KUKA KRL program: MyProgram_027().src

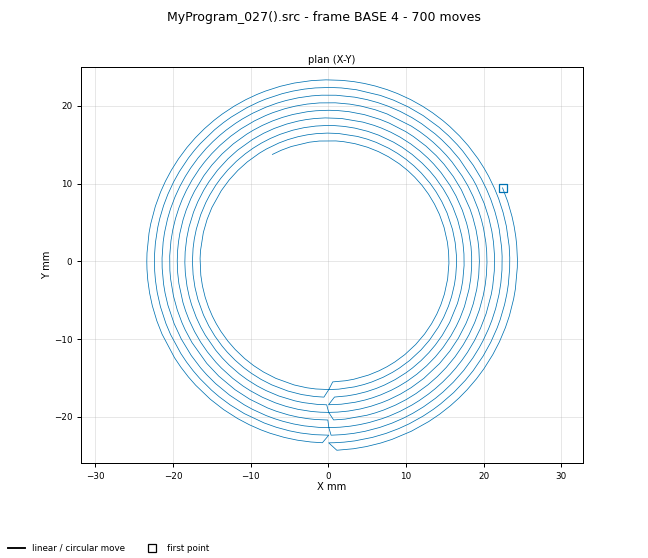
[picture p0: tool path of MyProgram_027().src in frame BASE 4, 700 of 700 moves have a stored position in this frame; points joined in program order, loops and branches not executed]
&ACCESS RVP
&REL 1
&PARAM TEMPLATE = C:\KRC\Roboter\Template\vorgabe
&PARAM EDITMASK = *
DEF MyProgram_027()
; ---- Setting reference (Base) ----
$BASE = BASE_DATA[4]

; --------------------------
; ---- Setting tool (TCP) ----
$TOOL = TOOL_DATA[3]
; --------------------------

$VEL.CP = VEL_APROX_PRINT
Startdeposition()
$VEL.CP = VEL_PRINT
LIN {X 22.4287,Y 9.4564,Z 58,A 14.1912,B 24.8124,C -3.1589,E1 25.1485,E2 -651.5768} C_DIS
LIN {X 23.1014,Y 7.6686,Z 58,A 9.7649,B 24.8138,C -3.1468,E1 25.1526,E2 -647.1466} C_DIS
LIN {X 23.6458,Y 5.7738,Z 58,A 5.5518,B 24.8149,C -3.1377,E1 25.1557,E2 -642.9363} C_DIS
LIN {X 23.9173,Y 4.5201,Z 58,A 2.5126,B 24.816,C -3.1284,E1 25.1574,E2 -639.8928} C_DIS
LIN {X 24.1337,Y 3.1677,Z 58,A -0.5395,B 24.8169,C -3.1205,E1 25.1586,E2 -636.8398} C_DIS
LIN {X 24.2489,Y 2.1152,Z 58,A -3.4554,B 24.8184,C -3.1081,E1 25.1594,E2 -633.9119} C_DIS
LIN {X 24.3395,Y 0.2898,Z 58,A -7.2887,B 24.8193,C -3.0999,E1 25.1598,E2 -630.082} C_DIS
LIN {X 24.3283,Y -0.7779,Z 58,A -10.7104,B 24.8214,C -3.082,E1 25.1595,E2 -626.6383} C_DIS
LIN {X 24.0781,Y -3.5664,Z 58,A -15.9759,B 24.8221,C -3.0762,E1 25.158,E2 -621.39} C_DIS
LIN {X 23.8573,Y -4.8272,Z 58,A -20.0449,B 24.8245,C -3.0551,E1 25.1558,E2 -617.295} C_DIS
LIN {X 23.313,Y -6.9977,Z 58,A -24.788,B 24.8257,C -3.0447,E1 25.1524,E2 -612.5545} C_DIS
LIN {X 22.7904,Y -8.5482,Z 58,A -28.7704,B 24.8272,C -3.0317,E1 25.1486,E2 -608.5636} C_DIS
LIN {X 22.0222,Y -10.3681,Z 58,A -33.8022,B 24.8293,C -3.0139,E1 25.1429,E2 -603.517} C_DIS
LIN {X 21.1792,Y -11.9952,Z 58,A -37.9863,B 24.8305,C -3.003,E1 25.1373,E2 -599.3291} C_DIS
LIN {X 20.022,Y -13.8417,Z 58,A -42.6404,B 24.8315,C -2.9941,E1 25.1302,E2 -594.677} C_DIS
LIN {X 19.0636,Y -15.1342,Z 58,A -46.5415,B 24.8328,C -2.983,E1 25.1235,E2 -590.7681} C_DIS
LIN {X 17.8586,Y -16.5394,Z 58,A -50.7568,B 24.8338,C -2.9737,E1 25.1157,E2 -586.5496} C_DIS
LIN {X 16.8309,Y -17.584,Z 58,A -54.1448,B 24.8346,C -2.9662,E1 25.109,E2 -583.1581} C_DIS
LIN {X 15.7146,Y -18.588,Z 58,A -57.8818,B 24.8358,C -2.9563,E1 25.1011,E2 -579.4124} C_DIS
LIN {X 14.3281,Y -19.6766,Z 58,A -61.9971,B 24.8367,C -2.9481,E1 25.0919,E2 -575.2925} C_DIS
LIN {X 12.9267,Y -20.6245,Z 58,A -66.2083,B 24.8377,C -2.9384,E1 25.082,E2 -571.072} C_DIS
LIN {X 10.6726,Y -21.8765,Z 58,A -72.7265,B 24.8393,C -2.9241,E1 25.0658,E2 -564.5382} C_DIS
LIN {X 8.2202,Y -22.9104,Z 58,A -78.0666,B 24.8393,C -2.9242,E1 25.052,E2 -559.2102} C_DIS
LIN {X 6.7478,Y -23.3869,Z 58,A -81.784,B 24.8398,C -2.9194,E1 25.0421,E2 -555.488} C_DIS
LIN {X 4.9064,Y -23.841,Z 58,A -86.3778,B 24.8404,C -2.9142,E1 25.0295,E2 -550.888} C_DIS
LIN {X 3.2399,Y -24.124,Z 58,A -90.0318,B 24.8404,C -2.9142,E1 25.0195,E2 -547.2376} C_DIS
LIN {X 1.0965,Y -24.316,Z 58,A -95.7147,B 24.8412,C -2.9068,E1 25.0036,E2 -541.5396} C_DIS
LIN {X 1.0965,Y -24.316,Z 58,A -95.7147,B 24.8412,C -2.9068,E1 25.0036,E2 -541.5396} C_DIS
Enddeposition()
LIN {X 0.0491,Y -23.3612,Z 58,A -97.7933,B 24.839,C -2.9266,E1 24.9979,E2 -539.5083} C_DIS
Startdeposition()
$VEL.CP = VEL_PRINT
LIN {X 0.753,Y -23.3494,Z 58,A -94.2208,B 24.8374,C -2.9419,E1 25.008,E2 -543.1168} C_DIS
LIN {X 2.0258,Y -23.2738,Z 58,A -91.3521,B 24.8374,C -2.9412,E1 25.016,E2 -545.9823} C_DIS
LIN {X 3.4162,Y -23.1102,Z 58,A -87.1337,B 24.8364,C -2.9501,E1 25.0277,E2 -550.2184} C_DIS
LIN {X 5.6877,Y -22.6583,Z 58,A -81.8177,B 24.8362,C -2.952,E1 25.0422,E2 -555.5318} C_DIS
LIN {X 7.425,Y -22.15,Z 58,A -77.4169,B 24.8357,C -2.9568,E1 25.0539,E2 -559.9358} C_DIS
LIN {X 9.059,Y -21.533,Z 58,A -73.7377,B 24.8357,C -2.957,E1 25.0634,E2 -563.6074} C_DIS
LIN {X 10.4154,Y -20.9112,Z 58,A -69.2878,B 24.8342,C -2.9701,E1 25.0747,E2 -568.0768} C_DIS
LIN {X 12.2027,Y -19.9213,Z 58,A -64.5258,B 24.8335,C -2.9765,E1 25.0862,E2 -572.8396} C_DIS
LIN {X 13.4975,Y -19.0679,Z 58,A -60.5918,B 24.8325,C -2.9852,E1 25.0953,E2 -576.7809} C_DIS
LIN {X 14.4357,Y -18.3677,Z 58,A -57.4005,B 24.8315,C -2.9945,E1 25.1023,E2 -579.9824} C_DIS
LIN {X 16.1336,Y -16.8961,Z 58,A -52.2089,B 24.8304,C -3.0037,E1 25.113,E2 -585.1748} C_DIS
LIN {X 17.6418,Y -15.3144,Z 58,A -47.4897,B 24.8297,C -3.0102,E1 25.1219,E2 -589.8886} C_DIS
LIN {X 18.6459,Y -14.0745,Z 58,A -42.8116,B 24.8276,C -3.0283,E1 25.13,E2 -594.5878} C_DIS
LIN {X 19.9336,Y -12.1826,Z 58,A -37.1639,B 24.8258,C -3.0441,E1 25.1386,E2 -600.2444} C_DIS
LIN {X 20.9152,Y -10.4066,Z 58,A -32.457,B 24.8245,C -3.0554,E1 25.1446,E2 -604.9534} C_DIS
LIN {X 21.729,Y -8.5794,Z 58,A -28.1395,B 24.8236,C -3.0635,E1 25.1494,E2 -609.2665} C_DIS
LIN {X 22.1157,Y -7.5274,Z 58,A -25.0112,B 24.8221,C -3.076,E1 25.1522,E2 -612.4065} C_DIS
LIN {X 22.6865,Y -5.5752,Z 58,A -20.1081,B 24.8205,C -3.0903,E1 25.1558,E2 -617.3155} C_DIS
LIN {X 22.9834,Y -4.1863,Z 58,A -16.5509,B 24.8191,C -3.1019,E1 25.1577,E2 -620.8794} C_DIS
LIN {X 23.1698,Y -2.9863,Z 58,A -13.4153,B 24.8178,C -3.1129,E1 25.1589,E2 -624.0226} C_DIS
LIN {X 23.3426,Y -0.9395,Z 58,A -8.919,B 24.8167,C -3.1227,E1 25.1597,E2 -628.5154} C_DIS
LIN {X 23.3568,Y 0.4688,Z 58,A -5.3427,B 24.8152,C -3.1348,E1 25.1597,E2 -632.0991} C_DIS
LIN {X 23.2798,Y 1.9538,Z 58,A -1.238,B 24.8133,C -3.1511,E1 25.1588,E2 -636.218} C_DIS
LIN {X 22.9166,Y 4.5391,Z 58,A 4.2783,B 24.8121,C -3.1609,E1 25.1564,E2 -641.7252} C_DIS
LIN {X 22.4933,Y 6.31,Z 58,A 9.6251,B 24.8094,C -3.1837,E1 25.1527,E2 -647.0951} C_DIS
LIN {X 21.9201,Y 8.0793,Z 58,A 13.523,B 24.8087,C -3.1897,E1 25.1491,E2 -650.9852} C_DIS
LIN {X 21.3892,Y 9.3949,Z 58,A 17.0683,B 24.8074,C -3.2001,E1 25.1452,E2 -654.5357} C_DIS
LIN {X 20.6396,Y 10.9433,Z 58,A 21.0402,B 24.8064,C -3.2088,E1 25.1403,E2 -658.5072} C_DIS
LIN {X 20.0488,Y 11.992,Z 58,A 24.1699,B 24.8052,C -3.2183,E1 25.1359,E2 -661.6433} C_DIS
LIN {X 19.2723,Y 13.2041,Z 58,A 28.0452,B 24.8037,C -3.2306,E1 25.1298,E2 -665.5285} C_DIS
LIN {X 18.0172,Y 14.871,Z 58,A 32.6958,B 24.8028,C -3.2378,E1 25.1218,E2 -670.1742} C_DIS
LIN {X 16.8934,Y 16.1364,Z 58,A 37.2521,B 24.8012,C -3.2508,E1 25.1132,E2 -674.7413} C_DIS
LIN {X 15.6106,Y 17.3802,Z 58,A 41.0651,B 24.8008,C -3.2539,E1 25.1054,E2 -678.5461} C_DIS
LIN {X 14.7291,Y 18.1332,Z 58,A 44.1503,B 24.7999,C -3.2614,E1 25.0988,E2 -681.6374} C_DIS
LIN {X 13.4156,Y 19.1256,Z 58,A 48.0828,B 24.7992,C -3.2672,E1 25.0899,E2 -685.5697} C_DIS
LIN {X 12.1321,Y 19.9642,Z 58,A 51.8621,B 24.7985,C -3.273,E1 25.081,E2 -689.3507} C_DIS
LIN {X 10.5843,Y 20.8263,Z 58,A 56.5365,B 24.7974,C -3.2816,E1 25.0694,E2 -694.0322} C_DIS
LIN {X 8.9243,Y 21.5896,Z 58,A 60.8731,B 24.797,C -3.2851,E1 25.0583,E2 -698.3666} C_DIS
LIN {X 7.5693,Y 22.1011,Z 58,A 64.2683,B 24.7968,C -3.2868,E1 25.0494,E2 -701.7589} C_DIS
LIN {X 6.0229,Y 22.5716,Z 58,A 68.0624,B 24.7966,C -3.288,E1 25.0393,E2 -705.5495} C_DIS
LIN {X 4.6413,Y 22.8959,Z 58,A 71.552,B 24.7964,C -3.2897,E1 25.0297,E2 -709.0387} C_DIS
LIN {X 3.3103,Y 23.1258,Z 58,A 74.9008,B 24.7963,C -3.291,E1 25.0205,E2 -712.3873} C_DIS
LIN {X 1.8029,Y 23.2918,Z 58,A 79.0541,B 24.7958,C -3.2947,E1 25.0089,E2 -716.5471} C_DIS
LIN {X -0.2978,Y 23.3597,Z 58,A 84.0444,B 24.796,C -3.2926,E1 24.995,E2 -721.5319} C_DIS
LIN {X -2.16,Y 23.2614,Z 58,A 88.9205,B 24.796,C -3.2929,E1 24.9814,E2 -726.4107} C_DIS
LIN {X -4.3701,Y 22.9492,Z 58,A 94.1198,B 24.7967,C -3.2872,E1 24.9671,E2 -731.601} C_DIS
LIN {X -6.1836,Y 22.5282,Z 58,A 98.7838,B 24.7972,C -3.2835,E1 24.9545,E2 -736.263} C_DIS
LIN {X -8.1141,Y 21.9067,Z 58,A 103.4711,B 24.7982,C -3.2757,E1 24.9422,E2 -740.9406} C_DIS
LIN {X -9.2066,Y 21.4713,Z 58,A 106.4345,B 24.7986,C -3.2722,E1 24.9345,E2 -743.9025} C_DIS
LIN {X -10.609,Y 20.8137,Z 58,A 110.0922,B 24.7994,C -3.2655,E1 24.9254,E2 -747.5537} C_DIS
LIN {X -12.0964,Y 19.9859,Z 58,A 114.7123,B 24.8,C -3.2609,E1 24.9142,E2 -752.1767} C_DIS
LIN {X -13.6533,Y 18.9565,Z 58,A 118.5178,B 24.8016,C -3.2477,E1 24.9055,E2 -755.9633} C_DIS
LIN {X -14.6701,Y 18.1811,Z 58,A 122.2839,B 24.802,C -3.2447,E1 24.8972,E2 -759.7362} C_DIS
LIN {X -15.9382,Y 17.0802,Z 58,A 126.4482,B 24.8031,C -3.2358,E1 24.8886,E2 -763.8958} C_DIS
LIN {X -17.1134,Y 15.9031,Z 58,A 130.3724,B 24.8044,C -3.2253,E1 24.881,E2 -767.8117} C_DIS
LIN {X -18.1978,Y 14.649,Z 58,A 134.5254,B 24.8055,C -3.2155,E1 24.8736,E2 -771.9605} C_DIS
LIN {X -19.2941,Y 13.1713,Z 58,A 139.5365,B 24.8067,C -3.2061,E1 24.8655,E2 -776.9735} C_DIS
LIN {X -20.1991,Y 11.7375,Z 58,A 143.4691,B 24.8082,C -3.1934,E1 24.8599,E2 -780.8961} C_DIS
LIN {X -20.9677,Y 10.3014,Z 58,A 147.0142,B 24.8099,C -3.1798,E1 24.8554,E2 -784.4276} C_DIS
LIN {X -21.5908,Y 8.9216,Z 58,A 151.509,B 24.8107,C -3.1727,E1 24.8504,E2 -788.9301} C_DIS
LIN {X -22.265,Y 7.0731,Z 58,A 156.3218,B 24.8125,C -3.1581,E1 24.8461,E2 -793.7354} C_DIS
LIN {X -22.8563,Y 4.8334,Z 58,A 161.8894,B 24.8146,C -3.1401,E1 24.8425,E2 -799.2925} C_DIS
LIN {X -23.0779,Y 3.6294,Z 58,A 165.278,B 24.8155,C -3.1326,E1 24.8411,E2 -802.6833} C_DIS
LIN {X -23.337,Y 1.0643,Z 58,A 170.5929,B 24.8184,C -3.1082,E1 24.8399,E2 -807.9716} C_DIS
LIN {X -23.3617,Y -0.0144,Z 58,A 173.2645,B 24.8193,C -3.1,E1 24.8398,E2 -810.6398} C_DIS
LIN {X -23.3392,Y -1.02,Z 58,A 175.8052,B 24.8202,C -3.0927,E1 24.84,E2 -813.1783} C_DIS
LIN {X -23.2364,Y -2.414,Z 58,A 179.6817,B 24.8212,C -3.0843,E1 24.841,E2 -817.0578} C_DIS
LIN {X -23.0029,Y -4.0772,Z 58,A -176.121,B 24.8226,C -3.0721,E1 24.8428,E2 -821.251} C_DIS
LIN {X -22.6514,Y -5.7166,Z 58,A -171.9113,B 24.8239,C -3.0603,E1 24.8455,E2 -825.4571} C_DIS
LIN {X -22.0687,Y -7.664,Z 58,A -166.7853,B 24.8255,C -3.0466,E1 24.8499,E2 -830.5795} C_DIS
LIN {X -21.4015,Y -9.3668,Z 58,A -161.5782,B 24.8265,C -3.0378,E1 24.8556,E2 -835.7944} C_DIS
LIN {X -19.7861,Y -12.4207,Z 58,A -154.6271,B 24.83,C -3.0077,E1 24.865,E2 -842.7098} C_DIS
LIN {X -18.9703,Y -13.6339,Z 58,A -150.229,B 24.8305,C -3.0033,E1 24.872,E2 -847.1192} C_DIS
LIN {X -18.0166,Y -14.8715,Z 58,A -146.7524,B 24.8317,C -2.9925,E1 24.8781,E2 -850.5863} C_DIS
LIN {X -17.0625,Y -15.9571,Z 58,A -142.5184,B 24.8321,C -2.9888,E1 24.8861,E2 -854.8302} C_DIS
LIN {X -15.1815,Y -17.7562,Z 58,A -136.8493,B 24.834,C -2.9722,E1 24.8977,E2 -860.4824} C_DIS
LIN {X -13.4696,Y -19.0872,Z 58,A -130.4927,B 24.8343,C -2.9697,E1 24.912,E2 -866.8557} C_DIS
LIN {X -11.6792,Y -20.2323,Z 58,A -126.0931,B 24.8357,C -2.957,E1 24.9224,E2 -871.2386} C_DIS
LIN {X -10.1604,Y -21.0363,Z 58,A -122.0125,B 24.8363,C -2.951,E1 24.9326,E2 -875.3159} C_DIS
LIN {X -8.6852,Y -21.6874,Z 58,A -118.3884,B 24.837,C -2.9447,E1 24.9418,E2 -878.9333} C_DIS
LIN {X -7.4925,Y -22.1274,Z 58,A -114.5721,B 24.8368,C -2.947,E1 24.9519,E2 -882.7627} C_DIS
LIN {X -5.6895,Y -22.6585,Z 58,A -110.4971,B 24.8375,C -2.9403,E1 24.9629,E2 -886.8281} C_DIS
LIN {X -4.0034,Y -23.0159,Z 58,A -105.4321,B 24.837,C -2.945,E1 24.9768,E2 -891.9099} C_DIS
LIN {X -2.2388,Y -23.2541,Z 58,A -101.6737,B 24.8376,C -2.9397,E1 24.9872,E2 -895.6581} C_DIS
LIN {X -0.7601,Y -23.3492,Z 58,A -97.8291,B 24.8374,C -2.9417,E1 24.9979,E2 -899.5083} C_DIS
LIN {X -0.7601,Y -23.3492,Z 58,A -97.8291,B 24.8374,C -2.9417,E1 24.9979,E2 -899.5083} C_DIS
Enddeposition()
LIN {X 0.0594,Y -22.3764,Z 58,A -97.5822,B 24.837,C -2.9453,E1 24.9986,E2 -899.7639} C_DIS
Startdeposition()
$VEL.CP = VEL_PRINT
LIN {X -1.7887,Y -22.3107,Z 58,A -102.6934,B 24.8373,C -2.9422,E1 24.9844,E2 -894.6438} C_DIS
LIN {X -3.5725,Y -22.0957,Z 58,A -107.3153,B 24.8373,C -2.943,E1 24.9716,E2 -890.0201} C_DIS
LIN {X -4.9833,Y -21.8206,Z 58,A -110.5248,B 24.8367,C -2.9478,E1 24.9628,E2 -886.8182} C_DIS
LIN {X -6.6868,Y -21.3602,Z 58,A -116.1215,B 24.8372,C -2.9436,E1 24.9478,E2 -881.2024} C_DIS
LIN {X -8.2481,Y -20.8072,Z 58,A -120.6031,B 24.8369,C -2.946,E1 24.9361,E2 -876.7169} C_DIS
LIN {X -10.8134,Y -19.5971,Z 58,A -126.9982,B 24.8353,C -2.96,E1 24.9202,E2 -870.3379} C_DIS
LIN {X -12.6262,Y -18.4813,Z 58,A -133.0282,B 24.8348,C -2.9649,E1 24.9061,E2 -864.3002} C_DIS
LIN {X -14.016,Y -17.4505,Z 58,A -136.4557,B 24.8333,C -2.9781,E1 24.8986,E2 -860.8916} C_DIS
LIN {X -15.0383,Y -16.5769,Z 58,A -140.5893,B 24.833,C -2.9809,E1 24.8899,E2 -856.7484} C_DIS
LIN {X -16.5556,Y -15.0627,Z 58,A -145.4598,B 24.8314,C -2.9955,E1 24.8805,E2 -851.8918} C_DIS
LIN {X -17.4052,Y -14.0722,Z 58,A -149.0695,B 24.8307,C -3.0017,E1 24.874,E2 -848.2803} C_DIS
LIN {X -18.2465,Y -12.9621,Z 58,A -152.5872,B 24.8297,C -3.0104,E1 24.8682,E2 -844.7665} C_DIS
LIN {X -18.9806,Y -11.8619,Z 58,A -156.8774,B 24.8292,C -3.0146,E1 24.8617,E2 -840.4647} C_DIS
LIN {X -20.3019,Y -9.4219,Z 58,A -163.3655,B 24.8267,C -3.0364,E1 24.8535,E2 -833.994} C_DIS
LIN {X -20.8927,Y -8.0277,Z 58,A -167.7212,B 24.8257,C -3.0452,E1 24.849,E2 -829.6351} C_DIS
LIN {X -21.613,Y -5.8178,Z 58,A -172.7995,B 24.8232,C -3.0663,E1 24.8449,E2 -824.5779} C_DIS
LIN {X -22.0246,Y -3.9859,Z 58,A -178.1948,B 24.8219,C -3.0782,E1 24.8418,E2 -819.1796} C_DIS
LIN {X -22.2472,Y -2.4581,Z 58,A 178.0676,B 24.8204,C -3.0912,E1 24.8405,E2 -815.4506} C_DIS
LIN {X -22.3486,Y -1.2274,Z 58,A 174.5283,B 24.8194,C -3.0994,E1 24.8399,E2 -811.9098} C_DIS
LIN {X -22.3659,Y 0.8536,Z 58,A 169.598,B 24.8173,C -3.1176,E1 24.8399,E2 -806.9933} C_DIS
LIN {X -22.2556,Y 2.3786,Z 58,A 165.1888,B 24.8161,C -3.1278,E1 24.8411,E2 -802.5821} C_DIS
LIN {X -21.9494,Y 4.382,Z 58,A 160.6412,B 24.8138,C -3.1465,E1 24.8432,E2 -798.0523} C_DIS
LIN {X -21.681,Y 5.5591,Z 58,A 157.1953,B 24.8129,C -3.1545,E1 24.8455,E2 -794.6055} C_DIS
LIN {X -21.2056,Y 7.1618,Z 58,A 152.9812,B 24.8113,C -3.1678,E1 24.849,E2 -790.3989} C_DIS
LIN {X -20.6553,Y 8.6217,Z 58,A 148.825,B 24.81,C -3.1789,E1 24.8533,E2 -786.2461} C_DIS
LIN {X -19.9176,Y 10.2106,Z 58,A 143.8606,B 24.8087,C -3.1898,E1 24.8593,E2 -781.281} C_DIS
LIN {X -19.1663,Y 11.5597,Z 58,A 139.9008,B 24.8073,C -3.2008,E1 24.865,E2 -777.3269} C_DIS
LIN {X -17.9987,Y 13.3051,Z 58,A 135.1411,B 24.8053,C -3.2178,E1 24.8725,E2 -772.5847} C_DIS
LIN {X -17.2488,Y 14.2633,Z 58,A 132.085,B 24.8043,C -3.2261,E1 24.8778,E2 -769.534} C_DIS
LIN {X -16.4585,Y 15.1687,Z 58,A 127.8731,B 24.804,C -3.2282,E1 24.8858,E2 -765.3085} C_DIS
LIN {X -14.6393,Y 16.9314,Z 58,A 122.0959,B 24.8018,C -3.2462,E1 24.8976,E2 -759.5511} C_DIS
LIN {X -13.4935,Y 17.8577,Z 58,A 118.4161,B 24.8008,C -3.2545,E1 24.9057,E2 -755.8775} C_DIS
LIN {X -12.501,Y 18.566,Z 58,A 114.5849,B 24.8005,C -3.2568,E1 24.9146,E2 -752.0389} C_DIS
LIN {X -10.4803,Y 19.7772,Z 58,A 109.1764,B 24.7988,C -3.2704,E1 24.9276,E2 -746.6472} C_DIS
LIN {X -9.0313,Y 20.4796,Z 58,A 105.3376,B 24.7978,C -3.2782,E1 24.9373,E2 -742.8173} C_DIS
LIN {X -8.0558,Y 20.8828,Z 58,A 101.9318,B 24.7979,C -3.2776,E1 24.9462,E2 -739.4028} C_DIS
LIN {X -5.9481,Y 21.5771,Z 58,A 96.8474,B 24.7967,C -3.2875,E1 24.9597,E2 -734.3332} C_DIS
LIN {X -4.5409,Y 21.9167,Z 58,A 92.9641,B 24.7964,C -3.2896,E1 24.9703,E2 -730.4499} C_DIS
LIN {X -3.0809,Y 22.1694,Z 58,A 89.0937,B 24.7962,C -3.2916,E1 24.981,E2 -726.5809} C_DIS
LIN {X -1.6805,Y 22.3194,Z 58,A 85.2928,B 24.7962,C -3.292,E1 24.9915,E2 -722.779} C_DIS
LIN {X 0.2375,Y 22.3811,Z 58,A 80.7154,B 24.7957,C -3.2955,E1 25.0043,E2 -718.2098} C_DIS
LIN {X 1.6744,Y 22.3198,Z 58,A 76.9456,B 24.7957,C -3.2949,E1 25.0148,E2 -714.44} C_DIS
LIN {X 3.6228,Y 22.0866,Z 58,A 70.9029,B 24.7969,C -3.2861,E1 25.0315,E2 -708.3818} C_DIS
LIN {X 6.6984,Y 21.3562,Z 58,A 63.2106,B 24.7971,C -3.2842,E1 25.0522,E2 -700.6972} C_DIS
LIN {X 8.4,Y 20.7463,Z 58,A 59.4451,B 24.7968,C -3.2869,E1 25.062,E2 -696.9462} C_DIS
LIN {X 10.3058,Y 19.8686,Z 58,A 52.692,B 24.799,C -3.2689,E1 25.079,E2 -690.1685} C_DIS
LIN {X 12.2114,Y 18.758,Z 58,A 47.4398,B 24.7996,C -3.2639,E1 25.0914,E2 -684.9211} C_DIS
LIN {X 14.2392,Y 17.269,Z 58,A 41.6217,B 24.8003,C -3.2582,E1 25.1042,E2 -679.1109} C_DIS
LIN {X 15.472,Y 16.1738,Z 58,A 37.5824,B 24.8011,C -3.2516,E1 25.1125,E2 -675.0722} C_DIS
LIN {X 16.6049,Y 15.0081,Z 58,A 33.7383,B 24.8019,C -3.2457,E1 25.1199,E2 -671.2309} C_DIS
LIN {X 17.3174,Y 14.1806,Z 58,A 30.4374,B 24.8032,C -3.2346,E1 25.1258,E2 -667.9188} C_DIS
LIN {X 18.6592,Y 12.3614,Z 58,A 24.2702,B 24.8054,C -3.2169,E1 25.1357,E2 -661.7396} C_DIS
LIN {X 19.684,Y 10.6539,Z 58,A 19.7371,B 24.8063,C -3.2091,E1 25.142,E2 -657.2117} C_DIS
LIN {X 20.3685,Y 9.2781,Z 58,A 16.0112,B 24.8074,C -3.2005,E1 25.1464,E2 -653.4853} C_DIS
LIN {X 20.9171,Y 7.9652,Z 58,A 12.3886,B 24.8086,C -3.1904,E1 25.1502,E2 -649.859} C_DIS
LIN {X 21.4372,Y 6.436,Z 58,A 8.0462,B 24.8103,C -3.1763,E1 25.1539,E2 -645.5077} C_DIS
LIN {X 21.7836,Y 5.1424,Z 58,A 5.1065,B 24.8109,C -3.1711,E1 25.1559,E2 -642.5728} C_DIS
LIN {X 21.9951,Y 4.1454,Z 58,A 1.6107,B 24.8129,C -3.1541,E1 25.1578,E2 -639.0571} C_DIS
LIN {X 22.3104,Y 1.7924,Z 58,A -3.5855,B 24.8141,C -3.1446,E1 25.1594,E2 -633.869} C_DIS
LIN {X 22.373,Y 0.6481,Z 58,A -6.8291,B 24.8155,C -3.1323,E1 25.1598,E2 -630.6154} C_DIS
LIN {X 22.3556,Y -1.1014,Z 58,A -10.8962,B 24.8167,C -3.1226,E1 25.1595,E2 -626.5495} C_DIS
LIN {X 22.2102,Y -2.7725,Z 58,A -15.339,B 24.8184,C -3.1076,E1 25.1582,E2 -622.0977} C_DIS
LIN {X 21.9749,Y -4.251,Z 58,A -19.4147,B 24.8201,C -3.0932,E1 25.1563,E2 -618.0116} C_DIS
LIN {X 21.5448,Y -6.0656,Z 58,A -23.856,B 24.8214,C -3.082,E1 25.1532,E2 -613.5693} C_DIS
LIN {X 21.0614,Y -7.5761,Z 58,A -28.0424,B 24.823,C -3.0684,E1 25.1495,E2 -609.3744} C_DIS
LIN {X 20.6289,Y -8.683,Z 58,A -31.1464,B 24.8241,C -3.0587,E1 25.1462,E2 -606.2646} C_DIS
LIN {X 19.9077,Y -10.2301,Z 58,A -35.0818,B 24.8251,C -3.0505,E1 25.1414,E2 -602.3309} C_DIS
LIN {X 19.4242,Y -11.1207,Z 58,A -38.0233,B 24.8263,C -3.0396,E1 25.1373,E2 -599.3789} C_DIS
LIN {X 18.6136,Y -12.4304,Z 58,A -42.1385,B 24.8278,C -3.0271,E1 25.1311,E2 -595.2547} C_DIS
LIN {X 17.4263,Y -14.0461,Z 58,A -46.9358,B 24.8289,C -3.017,E1 25.123,E2 -590.4562} C_DIS
LIN {X 16.0944,Y -15.554,Z 58,A -52.29,B 24.8306,C -3.0024,E1 25.1129,E2 -585.0911} C_DIS
LIN {X 14.7617,Y -16.824,Z 58,A -57.1683,B 24.832,C -2.9902,E1 25.1028,E2 -580.2034} C_DIS
LIN {X 13.7674,Y -17.6476,Z 58,A -60.2302,B 24.8325,C -2.9854,E1 25.0961,E2 -577.1417} C_DIS
LIN {X 12.2563,Y -18.7283,Z 58,A -65.0156,B 24.8336,C -2.9759,E1 25.085,E2 -572.35} C_DIS
LIN {X 10.8816,Y -19.5592,Z 58,A -68.887,B 24.8341,C -2.9708,E1 25.0757,E2 -568.4783} C_DIS
LIN {X 9.6925,Y -20.1748,Z 58,A -72.1113,B 24.8345,C -2.9672,E1 25.0676,E2 -565.254} C_DIS
LIN {X 8.1975,Y -20.8271,Z 58,A -77.0054,B 24.8359,C -2.9551,E1 25.055,E2 -560.3425} C_DIS
LIN {X 6.6205,Y -21.3808,Z 58,A -80.9282,B 24.8361,C -2.953,E1 25.0446,E2 -556.4223} C_DIS
LIN {X 4.7408,Y -21.8745,Z 58,A -86.0433,B 24.8368,C -2.9472,E1 25.0307,E2 -551.3005} C_DIS
LIN {X 3.2782,Y -22.1409,Z 58,A -89.3041,B 24.8366,C -2.9488,E1 25.0217,E2 -548.0468} C_DIS
LIN {X 1.843,Y -22.3064,Z 58,A -92.8669,B 24.8367,C -2.9478,E1 25.0118,E2 -544.4841} C_DIS
LIN {X 0.3571,Y -22.3795,Z 58,A -97.5689,B 24.8376,C -2.9398,E1 24.9986,E2 -539.7639} C_DIS
LIN {X 0.3571,Y -22.3795,Z 58,A -97.5689,B 24.8376,C -2.9398,E1 24.9986,E2 -539.7639} C_DIS
Enddeposition()
LIN {X 0.0693,Y -21.4022,Z 58,A -96.3339,B 24.8341,C -2.9713,E1 25.0023,E2 -541.074} C_DIS
Startdeposition()
$VEL.CP = VEL_PRINT
LIN {X 1.5198,Y -21.3493,Z 58,A -91.7701,B 24.8333,C -2.9779,E1 25.0151,E2 -545.652} C_DIS
LIN {X 2.8494,Y -21.2129,Z 58,A -88.6846,B 24.8335,C -2.9762,E1 25.0236,E2 -548.7311} C_DIS
LIN {X 4.0899,Y -21.0073,Z 58,A -85.405,B 24.8333,C -2.9782,E1 25.0326,E2 -552.0118} C_DIS
LIN {X 5.2662,Y -20.7452,Z 58,A -81.7581,B 24.8326,C -2.9846,E1 25.0425,E2 -555.6688} C_DIS
LIN {X 6.9059,Y -20.2584,Z 58,A -77.6775,B 24.8325,C -2.9857,E1 25.0534,E2 -559.7446} C_DIS
LIN {X 7.8829,Y -19.8986,Z 58,A -74.7362,B 24.8319,C -2.9907,E1 25.0611,E2 -562.6914} C_DIS
LIN {X 9.2231,Y -19.314,Z 58,A -70.3467,B 24.8308,C -3.0007,E1 25.0723,E2 -567.0936} C_DIS
LIN {X 10.7484,Y -18.5088,Z 58,A -66.2126,B 24.8304,C -3.0043,E1 25.0824,E2 -571.2242} C_DIS
LIN {X 11.7,Y -17.9216,Z 58,A -63.1037,B 24.8296,C -3.0109,E1 25.0897,E2 -574.3388} C_DIS
LIN {X 12.8554,Y -17.1124,Z 58,A -59.4843,B 24.8289,C -3.0171,E1 25.0979,E2 -577.9599} C_DIS
LIN {X 13.7488,Y -16.403,Z 58,A -56.3175,B 24.828,C -3.0247,E1 25.1048,E2 -581.1328} C_DIS
LIN {X 14.7388,Y -15.5201,Z 58,A -52.7543,B 24.8271,C -3.0329,E1 25.1121,E2 -584.701} C_DIS
LIN {X 15.6931,Y -14.5536,Z 58,A -49.3674,B 24.8264,C -3.0392,E1 25.1186,E2 -588.0883} C_DIS
LIN {X 16.4198,Y -13.7291,Z 58,A -46.2674,B 24.8253,C -3.0482,E1 25.1243,E2 -591.1954} C_DIS
LIN {X 17.2074,Y -12.7282,Z 58,A -42.9241,B 24.8244,C -3.0564,E1 25.1299,E2 -594.5423} C_DIS
LIN {X 17.9074,Y -11.7228,Z 58,A -39.2492,B 24.8229,C -3.0692,E1 25.1357,E2 -598.2294} C_DIS
LIN {X 18.8206,Y -10.1922,Z 58,A -34.6991,B 24.8216,C -3.0805,E1 25.142,E2 -602.7826} C_DIS
LIN {X 19.5937,Y -8.6123,Z 58,A -29.3344,B 24.8192,C -3.1009,E1 25.1482,E2 -608.1666} C_DIS
LIN {X 20.3118,Y -6.7471,Z 58,A -23.9701,B 24.8173,C -3.1171,E1 25.1532,E2 -613.5393} C_DIS
LIN {X 20.9731,Y -4.2692,Z 58,A -18.2317,B 24.8162,C -3.1266,E1 25.157,E2 -619.267} C_DIS
LIN {X 21.1564,Y -3.2408,Z 58,A -14.9725,B 24.8146,C -3.1401,E1 25.1584,E2 -622.5389} C_DIS
LIN {X 21.3682,Y -1.2241,Z 58,A -9.2908,B 24.8123,C -3.1597,E1 25.1597,E2 -628.2333} C_DIS
LIN {X 21.3873,Y 0.8276,Z 58,A -4.2264,B 24.8108,C -3.1723,E1 25.1595,E2 -633.2975} C_DIS
LIN {X 21.2582,Y 2.4869,Z 58,A 0.2319,B 24.8091,C -3.1861,E1 25.1583,E2 -637.7621} C_DIS
LIN {X 21.0478,Y 3.8847,Z 58,A 3.6058,B 24.8082,C -3.1934,E1 25.1567,E2 -641.1334} C_DIS
LIN {X 20.665,Y 5.5726,Z 58,A 9.342,B 24.8052,C -3.2183,E1 25.1528,E2 -646.8957} C_DIS
LIN {X 20.069,Y 7.4386,Z 58,A 14.4314,B 24.8036,C -3.2318,E1 25.1481,E2 -651.9884} C_DIS
LIN {X 19.0671,Y 9.7232,Z 58,A 19.9812,B 24.8027,C -3.2389,E1 25.1416,E2 -657.525} C_DIS
LIN {X 18.6099,Y 10.5724,Z 58,A 23.8934,B 24.8003,C -3.2586,E1 25.1361,E2 -661.4638} C_DIS
LIN {X 16.8781,Y 13.1612,Z 58,A 31.1716,B 24.799,C -3.2686,E1 25.1244,E2 -668.7301} C_DIS
LIN {X 15.6725,Y 14.5761,Z 58,A 36.4374,B 24.7973,C -3.2822,E1 25.1146,E2 -674.0048} C_DIS
LIN {X 14.6343,Y 15.6184,Z 58,A 40.2325,B 24.7965,C -3.2888,E1 25.107,E2 -677.7997} C_DIS
LIN {X 13.7487,Y 16.4035,Z 58,A 43.6494,B 24.7955,C -3.2969,E1 25.0997,E2 -681.2228} C_DIS
LIN {X 12.0117,Y 17.7147,Z 58,A 48.9825,B 24.7948,C -3.3023,E1 25.0876,E2 -686.5498} C_DIS
LIN {X 10.7598,Y 18.5017,Z 58,A 52.8179,B 24.7943,C -3.3069,E1 25.0785,E2 -690.3843} C_DIS
LIN {X 9.2573,Y 19.2976,Z 58,A 58.1125,B 24.7928,C -3.3187,E1 25.0652,E2 -695.6925} C_DIS
LIN {X 7.6976,Y 19.9713,Z 58,A 62.0521,B 24.7928,C -3.3182,E1 25.0551,E2 -699.6221} C_DIS
LIN {X 6.3869,Y 20.4277,Z 58,A 65.6538,B 24.7926,C -3.3203,E1 25.0455,E2 -703.2218} C_DIS
LIN {X 4.9912,Y 20.8132,Z 58,A 69.4819,B 24.7924,C -3.3222,E1 25.0352,E2 -707.0485} C_DIS
LIN {X 3.3995,Y 21.1316,Z 58,A 74.5674,B 24.7915,C -3.3293,E1 25.0212,E2 -712.1454} C_DIS
LIN {X 1.0071,Y 21.3796,Z 58,A 80.93,B 24.7915,C -3.329,E1 25.0035,E2 -718.5042} C_DIS
LIN {X -0.8511,Y 21.3863,Z 58,A 85.1036,B 24.7923,C -3.3223,E1 24.9919,E2 -722.662} C_DIS
LIN {X -2.12,Y 21.2982,Z 58,A 89.072,B 24.7921,C -3.3244,E1 24.9808,E2 -726.6375} C_DIS
LIN {X -3.8656,Y 21.0513,Z 58,A 93.663,B 24.7926,C -3.3204,E1 24.9682,E2 -731.2229} C_DIS
LIN {X -5.4449,Y 20.6991,Z 58,A 97.5083,B 24.7935,C -3.3134,E1 24.9578,E2 -735.057} C_DIS
LIN {X -6.6125,Y 20.3561,Z 58,A 101.0629,B 24.7937,C -3.3116,E1 24.9483,E2 -738.6134} C_DIS
LIN {X -8.0513,Y 19.8311,Z 58,A 105.4185,B 24.7942,C -3.3078,E1 24.9369,E2 -742.969} C_DIS
LIN {X -9.7406,Y 19.0582,Z 58,A 110.2465,B 24.7952,C -3.2994,E1 24.9248,E2 -747.7894} C_DIS
LIN {X -11.0483,Y 18.3307,Z 58,A 113.9019,B 24.7963,C -3.2906,E1 24.916,E2 -751.4348} C_DIS
LIN {X -11.947,Y 17.7586,Z 58,A 117.5019,B 24.7965,C -3.2892,E1 24.9076,E2 -755.0431} C_DIS
LIN {X -13.1313,Y 16.9018,Z 58,A 120.8139,B 24.7978,C -3.2782,E1 24.9002,E2 -758.3407} C_DIS
LIN {X -13.9343,Y 16.2461,Z 58,A 123.6422,B 24.7986,C -3.2725,E1 24.8942,E2 -761.1662} C_DIS
LIN {X -14.8529,Y 15.4106,Z 58,A 127.0044,B 24.7995,C -3.2652,E1 24.8873,E2 -764.5246} C_DIS
LIN {X -15.7184,Y 14.5269,Z 58,A 130.4415,B 24.8004,C -3.2578,E1 24.8807,E2 -767.9591} C_DIS
LIN {X -16.7726,Y 13.2957,Z 58,A 135.0521,B 24.8016,C -3.2481,E1 24.8725,E2 -772.5678} C_DIS
LIN {X -17.7086,Y 12.0208,Z 58,A 139.1812,B 24.803,C -3.2364,E1 24.8659,E2 -776.6891} C_DIS
LIN {X -18.4038,Y 10.927,Z 58,A 142.3461,B 24.8043,C -3.2256,E1 24.8613,E2 -779.8442} C_DIS
LIN {X -19.0851,Y 9.6879,Z 58,A 146.59,B 24.8054,C -3.2167,E1 24.8558,E2 -784.0896} C_DIS
LIN {X -19.7286,Y 8.2992,Z 58,A 150.5497,B 24.8069,C -3.2042,E1 24.8513,E2 -788.0409} C_DIS
LIN {X -20.3165,Y 6.7338,Z 58,A 154.7785,B 24.8087,C -3.1898,E1 24.8473,E2 -792.2592} C_DIS
LIN {X -20.6915,Y 5.474,Z 58,A 158.959,B 24.8096,C -3.1817,E1 24.8442,E2 -796.4446} C_DIS
LIN {X -21.0816,Y 3.6974,Z 58,A 163.3734,B 24.8116,C -3.1649,E1 24.8418,E2 -800.8446} C_DIS
LIN {X -21.2577,Y 2.4906,Z 58,A 167.1623,B 24.8126,C -3.1568,E1 24.8405,E2 -804.6369} C_DIS
LIN {X -21.3994,Y 0.402,Z 58,A 172.4761,B 24.8148,C -3.1382,E1 24.8398,E2 -809.938} C_DIS
LIN {X -21.3849,Y -0.8776,Z 58,A 176.3477,B 24.8159,C -3.1293,E1 24.8401,E2 -813.8118} C_DIS
LIN {X -21.2032,Y -2.9204,Z 58,A -178.7341,B 24.8181,C -3.1102,E1 24.8416,E2 -818.7135} C_DIS
LIN {X -21.0075,Y -4.0947,Z 58,A -175.2363,B 24.8191,C -3.1018,E1 24.8434,E2 -822.212} C_DIS
LIN {X -20.6458,Y -5.6437,Z 58,A -170.558,B 24.8204,C -3.091,E1 24.8466,E2 -826.8916} C_DIS
LIN {X -19.8389,Y -8.0321,Z 58,A -164.4138,B 24.8229,C -3.0691,E1 24.8524,E2 -833.0183} C_DIS
LIN {X -18.9192,Y -10.0068,Z 58,A -157.6316,B 24.8242,C -3.0576,E1 24.8608,E2 -839.8095} C_DIS
LIN {X -17.6345,Y -12.1284,Z 58,A -150.881,B 24.8261,C -3.0416,E1 24.8711,E2 -846.5558} C_DIS
LIN {X -16.4221,Y -13.7264,Z 58,A -146.525,B 24.8281,C -3.0243,E1 24.8786,E2 -850.8908} C_DIS
LIN {X -15.6668,Y -14.5823,Z 58,A -143.5566,B 24.8289,C -3.0173,E1 24.8842,E2 -853.8556} C_DIS
LIN {X -14.5057,Y -15.7379,Z 58,A -138.3999,B 24.8294,C -3.0125,E1 24.8946,E2 -859.0223} C_DIS
LIN {X -12.6922,Y -17.2334,Z 58,A -131.5397,B 24.8303,C -3.0047,E1 24.9097,E2 -865.8889} C_DIS
LIN {X -10.8237,Y -18.4648,Z 58,A -126.387,B 24.8318,C -2.9912,E1 24.9219,E2 -871.0254} C_DIS
LIN {X -9.7369,Y -19.0597,Z 58,A -122.9346,B 24.8322,C -2.9879,E1 24.9305,E2 -874.4794} C_DIS
LIN {X -7.9985,Y -19.8526,Z 58,A -118.2818,B 24.8331,C -2.9797,E1 24.9423,E2 -879.1238} C_DIS
LIN {X -6.9053,Y -20.2587,Z 58,A -115.1019,B 24.8334,C -2.9775,E1 24.9507,E2 -882.3047} C_DIS
LIN {X -5.8242,Y -20.5955,Z 58,A -112.1278,B 24.8337,C -2.9751,E1 24.9587,E2 -885.278} C_DIS
LIN {X -4.4547,Y -20.9347,Z 58,A -107.877,B 24.8335,C -2.9765,E1 24.9703,E2 -889.5376} C_DIS
LIN {X -3.0926,Y -21.1785,Z 58,A -104.2159,B 24.8336,C -2.9752,E1 24.9804,E2 -893.199} C_DIS
LIN {X -1.2575,Y -21.3663,Z 58,A -99.4586,B 24.8338,C -2.9737,E1 24.9936,E2 -897.955} C_DIS
LIN {X 0.0693,Y -21.4022,Z 58,A -97.6052,B 24.8351,C -2.962,E1 24.9987,E2 -899.7806} C_DIS
Enddeposition()
LIN {X 0.0693,Y -21.4022,Z 58,A -97.6052,B 24.8351,C -2.962,E1 24.9987,E2 -899.7806} C_DIS
Startdeposition()
$VEL.CP = VEL_PRINT
LIN {X -0.0586,Y -20.424,Z 58,A -98.287,B 24.8335,C -2.9769,E1 24.9969,E2 -899.1341} C_DIS
LIN {X -1.6552,Y -20.3567,Z 58,A -102.4124,B 24.8332,C -2.979,E1 24.9854,E2 -895.0127} C_DIS
LIN {X -2.7246,Y -20.2414,Z 58,A -105.6254,B 24.8333,C -2.9782,E1 24.9765,E2 -891.7956} C_DIS
LIN {X -3.9104,Y -20.0459,Z 58,A -108.963,B 24.8332,C -2.9795,E1 24.9673,E2 -888.4577} C_DIS
LIN {X -5.1213,Y -19.7715,Z 58,A -112.7276,B 24.8332,C -2.9796,E1 24.9571,E2 -884.6881} C_DIS
LIN {X -6.7102,Y -19.2901,Z 58,A -117.0919,B 24.8326,C -2.9848,E1 24.9455,E2 -880.3283} C_DIS
LIN {X -7.8166,Y -18.8693,Z 58,A -121.2762,B 24.8327,C -2.9831,E1 24.9346,E2 -876.1307} C_DIS
LIN {X -10.1008,Y -17.7516,Z 58,A -127.7286,B 24.8313,C -2.9956,E1 24.9187,E2 -869.6904} C_DIS
LIN {X -12.0003,Y -16.5256,Z 58,A -134.8567,B 24.8307,C -3.0016,E1 24.9022,E2 -862.5528} C_DIS
LIN {X -14.0953,Y -14.779,Z 58,A -143.2401,B 24.8294,C -3.0129,E1 24.8848,E2 -854.1631} C_DIS
LIN {X -15.6471,Y -13.1267,Z 58,A -149.7281,B 24.8278,C -3.0265,E1 24.873,E2 -847.678} C_DIS
LIN {X -17.5487,Y -10.4492,Z 58,A -157.6896,B 24.8246,C -3.0543,E1 24.8607,E2 -839.7431} C_DIS
LIN {X -18.4234,Y -8.8155,Z 58,A -162.3794,B 24.8228,C -3.0701,E1 24.8548,E2 -835.0663} C_DIS
LIN {X -18.8462,Y -7.8717,Z 58,A -165.7467,B 24.8221,C -3.0764,E1 24.851,E2 -831.6954} C_DIS
LIN {X -19.4425,Y -6.2548,Z 58,A -170.6189,B 24.8205,C -3.0901,E1 24.8466,E2 -826.8284} C_DIS
LIN {X -19.9345,Y -4.4434,Z 58,A -176.4767,B 24.8189,C -3.1037,E1 24.8427,E2 -820.9687} C_DIS
LIN {X -20.2972,Y -2.2732,Z 58,A 178.3183,B 24.8163,C -3.1258,E1 24.8406,E2 -815.7858} C_DIS
LIN {X -20.3898,Y -1.1818,Z 58,A 174.5621,B 24.8154,C -3.133,E1 24.8399,E2 -812.0242} C_DIS
LIN {X -20.412,Y 0.7019,Z 58,A 169.5522,B 24.8134,C -3.1504,E1 24.8399,E2 -807.0257} C_DIS
LIN {X -20.2541,Y 2.6291,Z 58,A 163.8252,B 24.8115,C -3.1662,E1 24.8416,E2 -801.3024} C_DIS
LIN {X -20.0148,Y 4.0678,Z 58,A 160.1309,B 24.8098,C -3.1802,E1 24.8435,E2 -797.6198} C_DIS
LIN {X -19.6661,Y 5.5125,Z 58,A 155.6043,B 24.8084,C -3.1917,E1 24.8466,E2 -793.0944} C_DIS
LIN {X -19.2249,Y 6.896,Z 58,A 151.7918,B 24.8068,C -3.2049,E1 24.8501,E2 -789.2918} C_DIS
LIN {X -18.7995,Y 7.9826,Z 58,A 148.612,B 24.8056,C -3.2149,E1 24.8534,E2 -786.1182} C_DIS
LIN {X -18.2634,Y 9.1429,Z 58,A 144.7735,B 24.8045,C -3.2244,E1 24.858,E2 -782.2815} C_DIS
LIN {X -17.5396,Y 10.4645,Z 58,A 140.2703,B 24.8031,C -3.2351,E1 24.8643,E2 -777.7806} C_DIS
LIN {X -16.5976,Y 11.9022,Z 58,A 135.8853,B 24.8014,C -3.2497,E1 24.8711,E2 -773.4089} C_DIS
LIN {X -15.9514,Y 12.7546,Z 58,A 132.6547,B 24.8005,C -3.2566,E1 24.8767,E2 -770.1793} C_DIS
LIN {X -15.0209,Y 13.8388,Z 58,A 128.7199,B 24.7993,C -3.2667,E1 24.884,E2 -766.2511} C_DIS
LIN {X -13.9341,Y 14.9327,Z 58,A 123.9175,B 24.7983,C -3.2746,E1 24.8936,E2 -761.4478} C_DIS
LIN {X -12.5691,Y 16.0986,Z 58,A 118.783,B 24.797,C -3.2849,E1 24.9047,E2 -756.3183} C_DIS
LIN {X -11.2286,Y 17.0604,Z 58,A 114.2023,B 24.7959,C -3.2939,E1 24.9152,E2 -751.744} C_DIS
LIN {X -9.4998,Y 18.0799,Z 58,A 108.6201,B 24.7947,C -3.3037,E1 24.9288,E2 -746.1689} C_DIS
LIN {X -8.069,Y 18.7626,Z 58,A 104.5369,B 24.7936,C -3.312,E1 24.9392,E2 -742.0955} C_DIS
LIN {X -7.1544,Y 19.1301,Z 58,A 101.811,B 24.7932,C -3.3158,E1 24.9463,E2 -739.3729} C_DIS
LIN {X -5.5628,Y 19.6518,Z 58,A 96.7663,B 24.7927,C -3.3191,E1 24.9597,E2 -734.3274} C_DIS
LIN {X -4.2156,Y 19.9843,Z 58,A 93.1762,B 24.7921,C -3.3242,E1 24.9695,E2 -730.7449} C_DIS
LIN {X -2.7291,Y 20.2411,Z 58,A 88.7078,B 24.7919,C -3.3257,E1 24.9818,E2 -726.2759} C_DIS
LIN {X -1.1362,Y 20.3923,Z 58,A 84.4361,B 24.7915,C -3.3289,E1 24.9937,E2 -722.0102} C_DIS
LIN {X 0.9095,Y 20.4035,Z 58,A 77.9916,B 24.792,C -3.3253,E1 25.0117,E2 -715.5578} C_DIS
LIN {X 2.7577,Y 20.237,Z 58,A 73.2176,B 24.7917,C -3.3273,E1 25.0249,E2 -710.7922} C_DIS
LIN {X 4.1986,Y 19.9878,Z 58,A 69.3564,B 24.7917,C -3.3273,E1 25.0355,E2 -706.9355} C_DIS
LIN {X 6.0293,Y 19.5136,Z 58,A 62.8077,B 24.7933,C -3.3149,E1 25.0531,E2 -700.3683} C_DIS
LIN {X 7.5645,Y 18.9717,Z 58,A 57.861,B 24.7942,C -3.3077,E1 25.0659,E2 -695.4154} C_DIS
LIN {X 10.6862,Y 17.4054,Z 58,A 49.5823,B 24.7942,C -3.3067,E1 25.0862,E2 -687.1582} C_DIS
LIN {X 11.811,Y 16.6626,Z 58,A 45.9738,B 24.7949,C -3.3021,E1 25.0945,E2 -683.551} C_DIS
LIN {X 12.7406,Y 15.9631,Z 58,A 42.64,B 24.7957,C -3.2958,E1 25.1019,E2 -680.2145} C_DIS
LIN {X 13.5152,Y 15.313,Z 58,A 39.9046,B 24.7962,C -3.2913,E1 25.1077,E2 -677.4792} C_DIS
LIN {X 14.4157,Y 14.4683,Z 58,A 36.4249,B 24.7971,C -3.2842,E1 25.1146,E2 -673.9971} C_DIS
LIN {X 15.1821,Y 13.6618,Z 58,A 33.4052,B 24.7978,C -3.2784,E1 25.1204,E2 -670.9767} C_DIS
LIN {X 15.9166,Y 12.7987,Z 58,A 29.4311,B 24.7996,C -3.2641,E1 25.1274,E2 -666.9872} C_DIS
LIN {X 17.2139,Y 10.9905,Z 58,A 24.0443,B 24.8005,C -3.2565,E1 25.1359,E2 -661.6089} C_DIS
LIN {X 17.9732,Y 9.7008,Z 58,A 19.3939,B 24.8024,C -3.2414,E1 25.1423,E2 -656.9469} C_DIS
LIN {X 18.6484,Y 8.3282,Z 58,A 15.4246,B 24.8034,C -3.2327,E1 25.147,E2 -652.9783} C_DIS
LIN {X 19.2972,Y 6.6905,Z 58,A 10.2572,B 24.8054,C -3.2165,E1 25.1521,E2 -647.8013} C_DIS
LIN {X 19.7221,Y 5.308,Z 58,A 6.6859,B 24.8063,C -3.2092,E1 25.1548,E2 -644.2332} C_DIS
LIN {X 19.978,Y 4.2461,Z 58,A 3.1372,B 24.808,C -3.1954,E1 25.157,E2 -640.6724} C_DIS
LIN {X 20.276,Y 2.4494,Z 58,A -1.2391,B 24.809,C -3.1869,E1 25.1588,E2 -636.3018} C_DIS
LIN {X 20.3868,Y 1.2368,Z 58,A -5.233,B 24.8109,C -3.1708,E1 25.1596,E2 -632.2932} C_DIS
LIN {X 20.4234,Y -0.1534,Z 58,A -9.1641,B 24.8124,C -3.1583,E1 25.1597,E2 -628.3561} C_DIS
LIN {X 20.3511,Y -1.7262,Z 58,A -13.3196,B 24.8138,C -3.1471,E1 25.159,E2 -624.1986} C_DIS
LIN {X 20.1927,Y -3.0652,Z 58,A -17.337,B 24.8154,C -3.133,E1 25.1574,E2 -620.1715} C_DIS
LIN {X 19.9444,Y -4.3967,Z 58,A -21.1286,B 24.8168,C -3.1214,E1 25.1552,E2 -616.3744} C_DIS
LIN {X 19.4429,Y -6.254,Z 58,A -26.3141,B 24.8185,C -3.1069,E1 25.1512,E2 -611.1844} C_DIS
LIN {X 18.8367,Y -7.8943,Z 58,A -31.3988,B 24.8204,C -3.0906,E1 25.146,E2 -606.0892} C_DIS
LIN {X 18.098,Y -9.4659,Z 58,A -35.9167,B 24.8217,C -3.0799,E1 25.1404,E2 -601.5701} C_DIS
LIN {X 17.357,Y -10.7646,Z 58,A -40.0643,B 24.823,C -3.0686,E1 25.1345,E2 -597.417} C_DIS
LIN {X 16.3275,Y -12.2698,Z 58,A -45.5176,B 24.8249,C -3.0519,E1 25.1256,E2 -591.9505} C_DIS
LIN {X 15.1825,Y -13.6614,Z 58,A -50.538,B 24.8263,C -3.0395,E1 25.1164,E2 -586.9236} C_DIS
LIN {X 14.0413,Y -14.8319,Z 58,A -54.7084,B 24.8271,C -3.0325,E1 25.1081,E2 -582.754} C_DIS
LIN {X 12.8084,Y -15.9082,Z 58,A -59.4689,B 24.8285,C -3.021,E1 25.098,E2 -577.9847} C_DIS
LIN {X 11.283,Y -17.024,Z 58,A -65.3247,B 24.8302,C -3.0059,E1 25.0845,E2 -572.113} C_DIS
LIN {X 10.0173,Y -17.7988,Z 58,A -69.041,B 24.8306,C -3.0023,E1 25.0755,E2 -568.3994} C_DIS
LIN {X 8.6238,Y -18.514,Z 58,A -73.1215,B 24.8311,C -2.998,E1 25.0653,E2 -564.3194} C_DIS
LIN {X 7.1212,Y -19.1425,Z 58,A -77.4334,B 24.8315,C -2.9938,E1 25.0541,E2 -560.0073} C_DIS
LIN {X 6.0369,Y -19.5114,Z 58,A -80.5366,B 24.8319,C -2.9908,E1 25.0459,E2 -556.903} C_DIS
LIN {X 4.9776,Y -19.808,Z 58,A -84.881,B 24.8333,C -2.9782,E1 25.034,E2 -552.5352} C_DIS
LIN {X 2.156,Y -20.3099,Z 58,A -91.8757,B 24.8331,C -2.9802,E1 25.0148,E2 -545.5519} C_DIS
LIN {X 0.6815,Y -20.4127,Z 58,A -96.1827,B 24.8334,C -2.9775,E1 25.0028,E2 -541.2399} C_DIS
LIN {X 0.6815,Y -20.4127,Z 58,A -96.1827,B 24.8334,C -2.9775,E1 25.0028,E2 -541.2399} C_DIS
Enddeposition()
LIN {X 0.0511,Y -19.4427,Z 58,A -96.9327,B 24.8307,C -3.0011,E1 25.0008,E2 -540.5461} C_DIS
Startdeposition()
$VEL.CP = VEL_PRINT
LIN {X 1.1836,Y -19.4075,Z 58,A -93.0113,B 24.8301,C -3.0061,E1 25.0118,E2 -544.4786} C_DIS
LIN {X 2.5778,Y -19.2733,Z 58,A -88.3887,B 24.8295,C -3.012,E1 25.0246,E2 -549.1118} C_DIS
LIN {X 4.1342,Y -19.0002,Z 58,A -84.103,B 24.8294,C -3.0131,E1 25.0364,E2 -553.3951} C_DIS
LIN {X 5.5122,Y -18.6471,Z 58,A -79.4726,B 24.8285,C -3.0208,E1 25.0489,E2 -558.0363} C_DIS
LIN {X 6.875,Y -18.1889,Z 58,A -75.5852,B 24.8282,C -3.0234,E1 25.0591,E2 -561.9219} C_DIS
LIN {X 7.8016,Y -17.8111,Z 58,A -72.3688,B 24.8275,C -3.0298,E1 25.0674,E2 -565.1458} C_DIS
LIN {X 9.2834,Y -17.0856,Z 58,A -67.9775,B 24.827,C -3.0338,E1 25.0783,E2 -569.5346} C_DIS
LIN {X 10.656,Y -16.2647,Z 58,A -62.6309,B 24.8254,C -3.0478,E1 25.091,E2 -574.8974} C_DIS
LIN {X 12.2999,Y -15.0593,Z 58,A -56.0081,B 24.8233,C -3.0657,E1 25.1056,E2 -581.5383} C_DIS
LIN {X 14.3084,Y -13.1667,Z 58,A -48.3346,B 24.8216,C -3.0808,E1 25.1207,E2 -589.215} C_DIS
LIN {X 15.6338,Y -11.5614,Z 58,A -41.8805,B 24.8194,C -3.0996,E1 25.1318,E2 -595.6834} C_DIS
LIN {X 16.7369,Y -9.8978,Z 58,A -36.3622,B 24.8179,C -3.1125,E1 25.1399,E2 -601.204} C_DIS
LIN {X 17.71,Y -8.0285,Z 58,A -30.8877,B 24.8166,C -3.1235,E1 25.1466,E2 -606.6754} C_DIS
LIN {X 18.2038,Y -6.8355,Z 58,A -26.9273,B 24.8151,C -3.1363,E1 25.1507,E2 -610.6441} C_DIS
LIN {X 18.6624,Y -5.4607,Z 58,A -22.4221,B 24.8132,C -3.1515,E1 25.1544,E2 -615.1598} C_DIS
LIN {X 19.1117,Y -3.5826,Z 58,A -16.8377,B 24.8113,C -3.1681,E1 25.1577,E2 -620.751} C_DIS
LIN {X 19.3618,Y -1.7944,Z 58,A -11.486,B 24.8092,C -3.1849,E1 25.1594,E2 -626.1111} C_DIS
LIN {X 19.445,Y 0.0155,Z 58,A -6.2661,B 24.8074,C -3.2004,E1 25.1597,E2 -631.3365} C_DIS
LIN {X 19.3816,Y 1.567,Z 58,A -2.172,B 24.8062,C -3.21,E1 25.1591,E2 -635.4289} C_DIS
LIN {X 19.2749,Y 2.5617,Z 58,A 1.049,B 24.8048,C -3.2216,E1 25.1579,E2 -638.6585} C_DIS
LIN {X 19.015,Y 4.0665,Z 58,A 5.6091,B 24.8031,C -3.2357,E1 25.1555,E2 -643.2255} C_DIS
LIN {X 18.5977,Y 5.6771,Z 58,A 10.1401,B 24.8017,C -3.2467,E1 25.1521,E2 -647.7564} C_DIS
LIN {X 18.2359,Y 6.7499,Z 58,A 14.4122,B 24.7995,C -3.265,E1 25.148,E2 -652.048} C_DIS
LIN {X 17.1222,Y 9.216,Z 58,A 21.0629,B 24.7983,C -3.2744,E1 25.14,E2 -658.6853} C_DIS
LIN {X 16.0974,Y 10.9076,Z 58,A 28.4751,B 24.7947,C -3.3033,E1 25.1288,E2 -666.1289} C_DIS
LIN {X 14.8999,Y 12.494,Z 58,A 32.921,B 24.7946,C -3.3044,E1 25.1211,E2 -670.5565} C_DIS
LIN {X 13.8919,Y 13.6056,Z 58,A 38.3055,B 24.7924,C -3.322,E1 25.1108,E2 -675.9595} C_DIS
LIN {X 12.5684,Y 14.837,Z 58,A 43.4184,B 24.7913,C -3.3303,E1 25.1,E2 -681.072} C_DIS
LIN {X 10.9572,Y 16.0637,Z 58,A 48.6701,B 24.7908,C -3.3345,E1 25.0882,E2 -686.3149} C_DIS
LIN {X 9.9672,Y 16.6961,Z 58,A 52.9551,B 24.7894,C -3.346,E1 25.0779,E2 -690.6139} C_DIS
LIN {X 7.8256,Y 17.8002,Z 58,A 59.3655,B 24.789,C -3.3491,E1 25.0618,E2 -697.0148} C_DIS
LIN {X 6.6244,Y 18.2817,Z 58,A 63.7567,B 24.788,C -3.3568,E1 25.0503,E2 -701.415} C_DIS
LIN {X 4.6344,Y 18.8845,Z 58,A 69.6453,B 24.7877,C -3.359,E1 25.0345,E2 -707.2993} C_DIS
LIN {X 2.667,Y 19.2609,Z 58,A 75.322,B 24.7877,C -3.3594,E1 25.0189,E2 -712.971} C_DIS
LIN {X 1.1916,Y 19.4085,Z 58,A 79.5076,B 24.7877,C -3.3584,E1 25.0072,E2 -717.1522} C_DIS
LIN {X 0.0345,Y 19.445,Z 58,A 83.1254,B 24.7877,C -3.3592,E1 24.9971,E2 -720.7715} C_DIS
LIN {X -1.6042,Y 19.3786,Z 58,A 87.6955,B 24.7881,C -3.3558,E1 24.9844,E2 -725.3349} C_DIS
LIN {X -2.7437,Y 19.2503,Z 58,A 91.6333,B 24.788,C -3.357,E1 24.9735,E2 -729.2786} C_DIS
LIN {X -4.5785,Y 18.8981,Z 58,A 96.4714,B 24.789,C -3.3487,E1 24.9603,E2 -734.1027} C_DIS
LIN {X -5.8945,Y 18.5284,Z 58,A 100.3789,B 24.7896,C -3.3438,E1 24.9499,E2 -738.005} C_DIS
LIN {X -7.1591,Y 18.079,Z 58,A 104.7139,B 24.79,C -3.3407,E1 24.9385,E2 -742.3415} C_DIS
LIN {X -8.5026,Y 17.4875,Z 58,A 109.0367,B 24.7908,C -3.3343,E1 24.9276,E2 -746.6597} C_DIS
LIN {X -9.6381,Y 16.8882,Z 58,A 112.6003,B 24.7918,C -3.327,E1 24.9189,E2 -750.2161} C_DIS
LIN {X -10.5087,Y 16.3606,Z 58,A 116.3044,B 24.792,C -3.3247,E1 24.9101,E2 -753.9266} C_DIS
LIN {X -12.216,Y 15.1285,Z 58,A 122.3153,B 24.7937,C -3.3112,E1 24.8968,E2 -759.9269} C_DIS
LIN {X -13.6742,Y 13.824,Z 58,A 128.2209,B 24.7953,C -3.2988,E1 24.8848,E2 -765.8268} C_DIS
LIN {X -14.9862,Y 12.3896,Z 58,A 134.5922,B 24.7967,C -3.2871,E1 24.8732,E2 -772.1991} C_DIS
LIN {X -16.0216,Y 11.0189,Z 58,A 139.5421,B 24.7985,C -3.2732,E1 24.8652,E2 -777.14} C_DIS
LIN {X -17.2205,Y 9.0303,Z 58,A 145.3295,B 24.8013,C -3.2503,E1 24.8572,E2 -782.9026} C_DIS
LIN {X -17.6923,Y 8.0679,Z 58,A 149.0521,B 24.8022,C -3.2431,E1 24.8528,E2 -786.6283} C_DIS
LIN {X -18.2897,Y 6.6024,Z 58,A 153.6133,B 24.8039,C -3.2289,E1 24.8483,E2 -791.181} C_DIS
LIN {X -18.6956,Y 5.3456,Z 58,A 157.5607,B 24.8053,C -3.2173,E1 24.8451,E2 -795.1234} C_DIS
LIN {X -19.1087,Y 3.6003,Z 58,A 162.7816,B 24.8073,C -3.2008,E1 24.842,E2 -800.3355} C_DIS
LIN {X -19.2849,Y 2.4879,Z 58,A 165.8909,B 24.8087,C -3.1898,E1 24.8408,E2 -803.437} C_DIS
LIN {X -19.3961,Y 1.3764,Z 58,A 169.2369,B 24.8099,C -3.1797,E1 24.84,E2 -806.7789} C_DIS
LIN {X -19.444,Y 0.0232,Z 58,A 173.0775,B 24.8114,C -3.1668,E1 24.8398,E2 -810.6118} C_DIS
LIN {X -19.3896,Y -1.4634,Z 58,A 178.4619,B 24.8126,C -3.1566,E1 24.8406,E2 -816.0041} C_DIS
LIN {X -19.232,Y -2.8701,Z 58,A -177.0421,B 24.814,C -3.145,E1 24.8424,E2 -820.4991} C_DIS
LIN {X -18.71,Y -5.2951,Z 58,A -170.8047,B 24.817,C -3.1195,E1 24.8465,E2 -826.7119} C_DIS
LIN {X -18.3698,Y -6.376,Z 58,A -167.2947,B 24.8181,C -3.1105,E1 24.8496,E2 -830.2203} C_DIS
LIN {X -17.9198,Y -7.5486,Z 58,A -163.3416,B 24.8192,C -3.1011,E1 24.8537,E2 -834.1729} C_DIS
LIN {X -17.2137,Y -9.0433,Z 58,A -158.4612,B 24.8207,C -3.088,E1 24.8598,E2 -839.0483} C_DIS
LIN {X -16.4201,Y -10.4157,Z 58,A -153.7724,B 24.8221,C -3.0762,E1 24.8666,E2 -843.7328} C_DIS
LIN {X -15.5668,Y -11.6521,Z 58,A -149.1598,B 24.8232,C -3.0664,E1 24.8741,E2 -848.3444} C_DIS
LIN {X -14.4446,Y -13.0176,Z 58,A -144.395,B 24.8248,C -3.0529,E1 24.8827,E2 -853.0987} C_DIS
LIN {X -13.7627,Y -13.7354,Z 58,A -140.8411,B 24.8252,C -3.0497,E1 24.8897,E2 -856.6601} C_DIS
LIN {X -12.3125,Y -15.0502,Z 58,A -135.2853,B 24.8265,C -3.0379,E1 24.9014,E2 -862.2095} C_DIS
LIN {X -10.9699,Y -16.0545,Z 58,A -130.7608,B 24.8277,C -3.0278,E1 24.9117,E2 -866.7257} C_DIS
LIN {X -10.0074,Y -16.6722,Z 58,A -127.0451,B 24.828,C -3.0247,E1 24.9205,E2 -870.4455} C_DIS
LIN {X -8.4675,Y -17.5044,Z 58,A -121.6326,B 24.8286,C -3.0197,E1 24.9339,E2 -875.8608} C_DIS
LIN {X -6.824,Y -18.2082,Z 58,A -116.2733,B 24.8291,C -3.0153,E1 24.9478,E2 -881.2212} C_DIS
LIN {X -5.431,Y -18.6712,Z 58,A -112.6105,B 24.8299,C -3.0084,E1 24.9576,E2 -884.8739} C_DIS
LIN {X -3.9101,Y -19.0476,Z 58,A -107.0325,B 24.8295,C -3.0121,E1 24.9728,E2 -890.4679} C_DIS
LIN {X -2.1729,Y -19.3232,Z 58,A -102.9987,B 24.8304,C -3.0037,E1 24.9839,E2 -894.485} C_DIS
LIN {X -0.9808,Y -19.42,Z 58,A -98.9508,B 24.83,C -3.0072,E1 24.9952,E2 -898.5426} C_DIS
LIN {X 0.0511,Y -19.4427,Z 58,A -96.9326,B 24.8307,C -3.001,E1 25.0008,E2 -900.5461} C_DIS
Enddeposition()
LIN {X 0.0511,Y -19.4427,Z 58,A -96.9326,B 24.8307,C -3.001,E1 25.0008,E2 -900.5461} C_DIS
Startdeposition()
$VEL.CP = VEL_PRINT
LIN {X -0.207,Y -18.4647,Z 58,A -98.8902,B 24.8296,C -3.0105,E1 24.9954,E2 -898.6111} C_DIS
LIN {X -1.4481,Y -18.4088,Z 58,A -102.8492,B 24.8297,C -3.0098,E1 24.9844,E2 -894.6491} C_DIS
LIN {X -3.2204,Y -18.1827,Z 58,A -108.3044,B 24.8295,C -3.0116,E1 24.9693,E2 -889.1935} C_DIS
LIN {X -4.3079,Y -17.9561,Z 58,A -111.9551,B 24.8295,C -3.0121,E1 24.9594,E2 -885.5394} C_DIS
LIN {X -6.3691,Y -17.3323,Z 58,A -119.1342,B 24.8292,C -3.0147,E1 24.9403,E2 -878.353} C_DIS
LIN {X -8.027,Y -16.6297,Z 58,A -124.0155,B 24.8281,C -3.0242,E1 24.928,E2 -873.4824} C_DIS
LIN {X -9.1743,Y -16.0254,Z 58,A -127.8617,B 24.8274,C -3.0302,E1 24.9185,E2 -869.6397} C_DIS
LIN {X -10.4295,Y -15.2383,Z 58,A -133.1703,B 24.827,C -3.0341,E1 24.9061,E2 -864.323} C_DIS
LIN {X -11.4158,Y -14.5142,Z 58,A -136.7279,B 24.8261,C -3.0416,E1 24.8983,E2 -860.7704} C_DIS
LIN {X -12.7676,Y -13.3406,Z 58,A -142.483,B 24.8249,C -3.0516,E1 24.8864,E2 -855.0159} C_DIS
LIN {X -13.6192,Y -12.4699,Z 58,A -145.8953,B 24.8239,C -3.061,E1 24.8799,E2 -851.6111} C_DIS
LIN {X -14.4929,Y -11.4427,Z 58,A -150.7789,B 24.8231,C -3.068,E1 24.8714,E2 -846.7215} C_DIS
LIN {X -15.8252,Y -9.5158,Z 58,A -157.0047,B 24.8205,C -3.0896,E1 24.8618,E2 -840.5162} C_DIS
LIN {X -16.4159,Y -8.4551,Z 58,A -161.1961,B 24.8195,C -3.0981,E1 24.8563,E2 -836.323} C_DIS
LIN {X -16.9934,Y -7.2254,Z 58,A -165.6022,B 24.8183,C -3.1091,E1 24.8513,E2 -831.919} C_DIS
LIN {X -17.5928,Y -5.6094,Z 58,A -170.019,B 24.8161,C -3.1273,E1 24.8472,E2 -827.5207} C_DIS
LIN {X -17.9045,Y -4.5172,Z 58,A -174.1338,B 24.8151,C -3.1358,E1 24.8441,E2 -823.4025} C_DIS
LIN {X -18.1858,Y -3.2032,Z 58,A -178.7568,B 24.8138,C -3.1471,E1 24.8416,E2 -818.7791} C_DIS
LIN {X -18.4026,Y -1.525,Z 58,A 176.0425,B 24.8118,C -3.1633,E1 24.8401,E2 -813.5862} C_DIS
LIN {X -18.4657,Y -0.1659,Z 58,A 172.0054,B 24.8102,C -3.1769,E1 24.8398,E2 -809.5574} C_DIS
LIN {X -18.424,Y 1.2393,Z 58,A 167.278,B 24.8087,C -3.1895,E1 24.8404,E2 -804.8317} C_DIS
LIN {X -18.222,Y 2.9902,Z 58,A 162.2639,B 24.8065,C -3.2078,E1 24.8423,E2 -799.8314} C_DIS
LIN {X -17.9291,Y 4.419,Z 58,A 157.0819,B 24.805,C -3.2198,E1 24.8455,E2 -794.6479} C_DIS
LIN {X -17.3522,Y 6.3152,Z 58,A 150.9858,B 24.8027,C -3.2385,E1 24.8508,E2 -788.5618} C_DIS
LIN {X -16.8084,Y 7.6459,Z 58,A 146.6897,B 24.8011,C -3.2521,E1 24.8555,E2 -784.2744} C_DIS
LIN {X -16.0272,Y 9.1712,Z 58,A 140.8864,B 24.7994,C -3.2656,E1 24.8633,E2 -778.473} C_DIS
LIN {X -15.3613,Y 10.2477,Z 58,A 137.3984,B 24.7979,C -3.2776,E1 24.8686,E2 -774.9961} C_DIS
LIN {X -14.2536,Y 11.7389,Z 58,A 131.2509,B 24.7962,C -3.2912,E1 24.8791,E2 -768.8521} C_DIS
LIN {X -12.9213,Y 13.1911,Z 58,A 124.6994,B 24.7946,C -3.3042,E1 24.8918,E2 -762.3035} C_DIS
LIN {X -11.6877,Y 14.2963,Z 58,A 119.3336,B 24.7933,C -3.3144,E1 24.9033,E2 -756.9416} C_DIS
LIN {X -9.7867,Y 15.6589,Z 58,A 112.8658,B 24.7912,C -3.3312,E1 24.9182,E2 -750.4925} C_DIS
LIN {X -8.325,Y 16.4825,Z 58,A 108.1577,B 24.7899,C -3.3419,E1 24.9298,E2 -745.7967} C_DIS
LIN {X -6.9544,Y 17.106,Z 58,A 102.8032,B 24.7894,C -3.3455,E1 24.9435,E2 -740.438} C_DIS
LIN {X -5.3605,Y 17.6707,Z 58,A 97.7277,B 24.7886,C -3.3523,E1 24.9569,E2 -735.3696} C_DIS
LIN {X -3.8878,Y 18.0518,Z 58,A 93.4444,B 24.7877,C -3.3588,E1 24.9685,E2 -731.0959} C_DIS
LIN {X -2.9065,Y 18.2357,Z 58,A 90.2866,B 24.7875,C -3.3607,E1 24.9772,E2 -727.9396} C_DIS
LIN {X -1.8116,Y 18.3768,Z 58,A 86.6642,B 24.7874,C -3.3615,E1 24.9873,E2 -724.3168} C_DIS
LIN {X -0.4018,Y 18.4614,Z 58,A 81.8486,B 24.7875,C -3.3605,E1 25.0007,E2 -719.4978} C_DIS
LIN {X 1.6805,Y 18.389,Z 58,A 74.3998,B 24.7883,C -3.3547,E1 25.0215,E2 -712.0385} C_DIS
LIN {X 4.456,Y 17.9201,Z 58,A 66.9984,B 24.7877,C -3.3593,E1 25.0417,E2 -704.6571} C_DIS
LIN {X 5.8476,Y 17.5153,Z 58,A 62.7636,B 24.7879,C -3.3578,E1 25.053,E2 -700.4262} C_DIS
LIN {X 6.8234,Y 17.1589,Z 58,A 59.301,B 24.7884,C -3.3532,E1 25.062,E2 -696.9602} C_DIS
LIN {X 8.0548,Y 16.6159,Z 58,A 55.1735,B 24.789,C -3.3488,E1 25.0724,E2 -692.8328} C_DIS
LIN {X 9.2457,Y 15.9843,Z 58,A 50.8061,B 24.7899,C -3.3419,E1 25.0831,E2 -688.4616} C_DIS
LIN {X 10.6153,Y 15.1097,Z 58,A 45.8143,B 24.7908,C -3.3343,E1 25.0947,E2 -683.4686} C_DIS
LIN {X 11.8477,Y 14.1638,Z 58,A 41.4701,B 24.7914,C -3.3294,E1 25.1042,E2 -679.129} C_DIS
LIN {X 12.8231,Y 13.2871,Z 58,A 37.3118,B 24.7925,C -3.3208,E1 25.1127,E2 -674.967} C_DIS
LIN {X 13.5564,Y 12.5384,Z 58,A 33.7098,B 24.7938,C -3.311,E1 25.1197,E2 -671.3575} C_DIS
LIN {X 14.5145,Y 11.4154,Z 58,A 28.8471,B 24.7953,C -3.2983,E1 25.1282,E2 -666.4871} C_DIS
LIN {X 15.6695,Y 9.7691,Z 58,A 23.4033,B 24.7964,C -3.2896,E1 25.1367,E2 -661.0495} C_DIS
LIN {X 16.4321,Y 8.424,Z 58,A 17.7221,B 24.7989,C -3.2693,E1 25.1443,E2 -655.3502} C_DIS
LIN {X 17.256,Y 6.5735,Z 58,A 11.8158,B 24.8007,C -3.2551,E1 25.1506,E2 -649.4426} C_DIS
LIN {X 17.8049,Y 4.8949,Z 58,A 6.8877,B 24.8021,C -3.244,E1 25.1546,E2 -644.5163} C_DIS
LIN {X 18.0507,Y 3.8929,Z 58,A 2.9981,B 24.804,C -3.2283,E1 25.157,E2 -640.612} C_DIS
LIN {X 18.368,Y 1.8932,Z 58,A -2.5404,B 24.8055,C -3.2158,E1 25.1591,E2 -635.0766} C_DIS
LIN {X 18.454,Y 0.6519,Z 58,A -6.6235,B 24.8072,C -3.2018,E1 25.1598,E2 -630.9846} C_DIS
LIN {X 18.4525,Y -0.7026,Z 58,A -10.4858,B 24.8084,C -3.1918,E1 25.1596,E2 -627.1216} C_DIS
LIN {X 18.3333,Y -2.2066,Z 58,A -15.1884,B 24.8102,C -3.177,E1 25.1584,E2 -622.4119} C_DIS
LIN {X 18.1098,Y -3.6056,Z 58,A -20.4819,B 24.8128,C -3.1553,E1 25.1557,E2 -617.0978} C_DIS
LIN {X 17.5245,Y -5.82,Z 58,A -27.2034,B 24.815,C -3.1371,E1 25.1504,E2 -610.3715} C_DIS
LIN {X 16.9678,Y -7.2854,Z 58,A -31.5951,B 24.8162,C -3.1269,E1 25.1458,E2 -605.9799} C_DIS
LIN {X 16.4768,Y -8.3349,Z 58,A -35.2715,B 24.8175,C -3.1158,E1 25.1413,E2 -602.2969} C_DIS
LIN {X 15.7794,Y -9.5912,Z 58,A -39.4056,B 24.8186,C -3.1061,E1 25.1356,E2 -598.1612} C_DIS
LIN {X 14.7913,Y -11.0543,Z 58,A -45.2527,B 24.8207,C -3.0882,E1 25.1262,E2 -592.3003} C_DIS
LIN {X 13.7864,Y -12.2847,Z 58,A -50.4383,B 24.8224,C -3.0737,E1 25.1168,E2 -587.1039} C_DIS
LIN {X 12.6462,Y -13.4556,Z 58,A -55.1847,B 24.8235,C -3.0645,E1 25.1073,E2 -582.3555} C_DIS
LIN {X 11.3958,Y -14.5298,Z 58,A -60.4438,B 24.8249,C -3.0523,E1 25.096,E2 -577.0876} C_DIS
LIN {X 10.142,Y -15.4311,Z 58,A -65.0522,B 24.8258,C -3.0444,E1 25.0853,E2 -572.4762} C_DIS
LIN {X 9.0454,Y -16.0985,Z 58,A -68.7616,B 24.8263,C -3.0395,E1 25.0764,E2 -568.7664} C_DIS
LIN {X 8.1041,Y -16.5925,Z 58,A -72.4835,B 24.8273,C -3.031,E1 25.0671,E2 -565.0344} C_DIS
LIN {X 6.7575,Y -17.1847,Z 58,A -76.8178,B 24.8278,C -3.0263,E1 25.0559,E2 -560.699} C_DIS
LIN {X 5.6932,Y -17.5661,Z 58,A -80.0069,B 24.8281,C -3.0244,E1 25.0475,E2 -557.5115} C_DIS
LIN {X 4.7153,Y -17.8537,Z 58,A -83.162,B 24.8284,C -3.0211,E1 25.039,E2 -554.3537} C_DIS
LIN {X 3.4808,Y -18.1346,Z 58,A -87.9586,B 24.8295,C -3.0118,E1 25.0258,E2 -549.5411} C_DIS
LIN {X 1.6655,Y -18.3904,Z 58,A -93.2013,B 24.8295,C -3.0114,E1 25.0113,E2 -544.3013} C_DIS
LIN {X 0.0327,Y -18.4602,Z 58,A -96.096,B 24.8282,C -3.0237,E1 25.0033,E2 -541.4366} C_DIS
Enddeposition()
LIN {X 0.0327,Y -18.4602,Z 58,A -96.096,B 24.8282,C -3.0237,E1 25.0033,E2 -541.4366} C_DIS
Startdeposition()
$VEL.CP = VEL_PRINT
LIN {X 0.7973,Y -17.4683,Z 58,A -93.4742,B 24.8261,C -3.0418,E1 25.0107,E2 -544.1007} C_DIS
LIN {X 2.383,Y -17.3231,Z 58,A -88.4714,B 24.8259,C -3.0434,E1 25.0246,E2 -549.1038} C_DIS
LIN {X 3.5289,Y -17.1267,Z 58,A -84.3298,B 24.8253,C -3.0487,E1 25.036,E2 -553.2532} C_DIS
LIN {X 4.8972,Y -16.7869,Z 58,A -79.8975,B 24.8249,C -3.0521,E1 25.048,E2 -557.6867} C_DIS
LIN {X 6.1704,Y -16.3616,Z 58,A -75.7235,B 24.8244,C -3.056,E1 25.0589,E2 -561.8616} C_DIS
LIN {X 7.2121,Y -15.93,Z 58,A -72.1222,B 24.8239,C -3.0607,E1 25.0682,E2 -565.4652} C_DIS
LIN {X 8.6057,Y -15.2224,Z 58,A -66.4253,B 24.8224,C -3.0735,E1 25.0823,E2 -571.1765} C_DIS
LIN {X 10.0042,Y -14.342,Z 58,A -61.5647,B 24.8217,C -3.0795,E1 25.0936,E2 -576.0352} C_DIS
LIN {X 10.8165,Y -13.7397,Z 58,A -57.8768,B 24.8206,C -3.0894,E1 25.1018,E2 -579.733} C_DIS
LIN {X 11.9486,Y -12.7675,Z 58,A -53.1016,B 24.8194,C -3.0994,E1 25.1117,E2 -584.5129} C_DIS
LIN {X 12.9505,Y -11.7495,Z 58,A -48.775,B 24.8184,C -3.1078,E1 25.12,E2 -588.8406} C_DIS
LIN {X 13.7788,Y -10.7645,Z 58,A -44.6204,B 24.8172,C -3.118,E1 25.1274,E2 -593.0002} C_DIS
LIN {X 14.671,Y -9.5151,Z 58,A -39.1765,B 24.8152,C -3.1351,E1 25.136,E2 -598.4578} C_DIS
LIN {X 15.6162,Y -7.8672,Z 58,A -31.8076,B 24.8119,C -3.1629,E1 25.1457,E2 -605.8538} C_DIS
LIN {X 16.6278,Y -5.4123,Z 58,A -24.0968,B 24.8098,C -3.18,E1 25.1532,E2 -613.5622} C_DIS
LIN {X 17.0609,Y -3.8332,Z 58,A -19.1416,B 24.8083,C -3.1928,E1 25.1566,E2 -618.5192} C_DIS
LIN {X 17.298,Y -2.5626,Z 58,A -14.5837,B 24.8063,C -3.2088,E1 25.1586,E2 -623.0883} C_DIS
LIN {X 17.4783,Y -0.535,Z 58,A -7.9718,B 24.8039,C -3.2291,E1 25.1598,E2 -629.709} C_DIS
LIN {X 17.4605,Y 0.9519,Z 58,A -3.7116,B 24.8027,C -3.2388,E1 25.1594,E2 -633.9667} C_DIS
LIN {X 17.3442,Y 2.2259,Z 58,A 0.7954,B 24.8008,C -3.2544,E1 25.158,E2 -638.4842} C_DIS
LIN {X 17.1723,Y 3.2996,Z 58,A 4.473,B 24.7993,C -3.2662,E1 25.1562,E2 -642.1682} C_DIS
LIN {X 16.6551,Y 5.3276,Z 58,A 11.7891,B 24.7963,C -3.2903,E1 25.1505,E2 -649.4996} C_DIS
LIN {X 16.0145,Y 7.0224,Z 58,A 17.0653,B 24.795,C -3.3012,E1 25.145,E2 -654.7726} C_DIS
LIN {X 15.4546,Y 8.1814,Z 58,A 20.905,B 24.794,C -3.3093,E1 25.1401,E2 -658.6111} C_DIS
LIN {X 14.7875,Y 9.3335,Z 58,A 25.7741,B 24.792,C -3.3247,E1 25.1331,E2 -663.4919} C_DIS
LIN {X 13.8128,Y 10.7232,Z 58,A 30.8319,B 24.7909,C -3.3339,E1 25.1247,E2 -668.547} C_DIS
LIN {X 13.084,Y 11.6008,Z 58,A 34.5764,B 24.7898,C -3.3423,E1 25.1179,E2 -672.2944} C_DIS
LIN {X 12.1105,Y 12.614,Z 58,A 39.723,B 24.7881,C -3.356,E1 25.1077,E2 -677.4518} C_DIS
LIN {X 10.7729,Y 13.7738,Z 58,A 44.7667,B 24.7875,C -3.3608,E1 25.0969,E2 -682.4878} C_DIS
LIN {X 9.53,Y 14.6616,Z 58,A 50.0264,B 24.7862,C -3.3707,E1 25.0848,E2 -687.7531} C_DIS
LIN {X 8.3982,Y 15.3379,Z 58,A 55.246,B 24.7846,C -3.383,E1 25.0721,E2 -692.9865} C_DIS
LIN {X 6.4929,Y 16.2367,Z 58,A 61.3828,B 24.7844,C -3.3851,E1 25.0564,E2 -699.1132} C_DIS
LIN {X 5.0601,Y 16.7384,Z 58,A 66.4605,B 24.7838,C -3.3896,E1 25.0429,E2 -704.1922} C_DIS
LIN {X 3.4202,Y 17.1489,Z 58,A 72.0919,B 24.7834,C -3.3929,E1 25.0276,E2 -709.8239} C_DIS
LIN {X 2.0691,Y 17.3636,Z 58,A 76.076,B 24.7836,C -3.391,E1 25.0166,E2 -713.7999} C_DIS
LIN {X 0.8473,Y 17.4657,Z 58,A 80.0931,B 24.7836,C -3.391,E1 25.0054,E2 -717.8155} C_DIS
LIN {X -0.2603,Y 17.4846,Z 58,A 83.7156,B 24.7837,C -3.3903,E1 24.9953,E2 -721.4361} C_DIS
LIN {X -1.6048,Y 17.4112,Z 58,A 87.9587,B 24.784,C -3.3877,E1 24.9835,E2 -725.6744} C_DIS
LIN {X -3.1229,Y 17.2054,Z 58,A 93.7713,B 24.784,C -3.3883,E1 24.9674,E2 -731.4937} C_DIS
LIN {X -4.5716,Y 16.8783,Z 58,A 98.6976,B 24.7845,C -3.384,E1 24.9541,E2 -736.4167} C_DIS
LIN {X -6.214,Y 16.3451,Z 58,A 103.7073,B 24.7858,C -3.3742,E1 24.9409,E2 -741.4128} C_DIS
LIN {X -7.4657,Y 15.8127,Z 58,A 108.5326,B 24.7864,C -3.3693,E1 24.9287,E2 -746.2381} C_DIS
LIN {X -8.606,Y 15.2224,Z 58,A 112.3992,B 24.7874,C -3.361,E1 24.9192,E2 -750.0957} C_DIS
LIN {X -9.6669,Y 14.5715,Z 58,A 116.8228,B 24.7882,C -3.3549,E1 24.9088,E2 -754.5189} C_DIS
LIN {X -10.6827,Y 13.844,Z 58,A 120.6241,B 24.7894,C -3.3455,E1 24.9003,E2 -758.3114} C_DIS
LIN {X -11.8339,Y 12.8737,Z 58,A 125.9666,B 24.7906,C -3.3362,E1 24.8891,E2 -763.6525} C_DIS
LIN {X -12.9284,Y 11.7745,Z 58,A 130.9462,B 24.7922,C -3.3237,E1 24.8795,E2 -768.6239} C_DIS
LIN {X -13.8577,Y 10.6647,Z 58,A 135.397,B 24.7938,C -3.3108,E1 24.8717,E2 -773.0644} C_DIS
LIN {X -14.4817,Y 9.8009,Z 58,A 139.2586,B 24.7948,C -3.3026,E1 24.8656,E2 -776.9255} C_DIS
LIN {X -15.252,Y 8.552,Z 58,A 143.6888,B 24.7966,C -3.2882,E1 24.8593,E2 -781.344} C_DIS
LIN {X -15.7627,Y 7.5706,Z 58,A 147.4419,B 24.7979,C -3.2781,E1 24.8546,E2 -785.0932} C_DIS
LIN {X -16.4198,Y 6.0138,Z 58,A 153.8593,B 24.7996,C -3.2642,E1 24.848,E2 -791.5131} C_DIS
LIN {X -16.9838,Y 4.1622,Z 58,A 159.6204,B 24.8021,C -3.2433,E1 24.8437,E2 -797.2575} C_DIS
LIN {X -17.2503,Y 2.8643,Z 58,A 164.0583,B 24.8038,C -3.2301,E1 24.8414,E2 -801.6902} C_DIS
LIN {X -17.4061,Y 1.6744,Z 58,A 168.1997,B 24.8052,C -3.2185,E1 24.8402,E2 -805.8283} C_DIS
LIN {X -17.4866,Y -0.0016,Z 58,A 173.8186,B 24.8072,C -3.2017,E1 24.8398,E2 -811.4409} C_DIS
LIN {X -17.402,Y -1.7152,Z 58,A 178.8791,B 24.8095,C -3.1828,E1 24.8408,E2 -816.4867} C_DIS
LIN {X -17.1666,Y -3.3294,Z 58,A -174.4748,B 24.811,C -3.1703,E1 24.8439,E2 -823.1421} C_DIS
LIN {X -16.7773,Y -4.9296,Z 58,A -169.1516,B 24.8129,C -3.1542,E1 24.848,E2 -828.4577} C_DIS
LIN {X -16.0681,Y -6.8994,Z 58,A -162.9684,B 24.8155,C -3.1329,E1 24.8542,E2 -834.6243} C_DIS
LIN {X -15.3838,Y -8.3135,Z 58,A -158.1285,B 24.8172,C -3.1182,E1 24.8603,E2 -839.455} C_DIS
LIN {X -14.5999,Y -9.6239,Z 58,A -152.1801,B 24.8183,C -3.1087,E1 24.8692,E2 -845.411} C_DIS
LIN {X -13.6518,Y -10.9274,Z 58,A -148.0124,B 24.8202,C -3.0925,E1 24.8762,E2 -849.5597} C_DIS
LIN {X -12.991,Y -11.7053,Z 58,A -143.973,B 24.8208,C -3.0877,E1 24.8837,E2 -853.6057} C_DIS
LIN {X -11.9884,Y -12.7301,Z 58,A -139.5441,B 24.822,C -3.0772,E1 24.8925,E2 -858.028} C_DIS
LIN {X -10.9096,Y -13.6662,Z 58,A -134.9963,B 24.823,C -3.0681,E1 24.9022,E2 -862.5716} C_DIS
LIN {X -9.8935,Y -14.417,Z 58,A -130.9813,B 24.8239,C -3.0608,E1 24.9113,E2 -866.5832} C_DIS
LIN {X -8.6419,Y -15.202,Z 58,A -125.4958,B 24.8243,C -3.0568,E1 24.9245,E2 -872.0759} C_DIS
LIN {X -7.2681,Y -15.9046,Z 58,A -119.9988,B 24.8248,C -3.0532,E1 24.9383,E2 -877.5783} C_DIS
LIN {X -5.1997,Y -16.695,Z 58,A -113.2925,B 24.8258,C -3.0444,E1 24.956,E2 -884.2769} C_DIS
LIN {X -3.4403,Y -17.1447,Z 58,A -107.2,B 24.826,C -3.0423,E1 24.9726,E2 -890.3723} C_DIS
LIN {X -1.8021,Y -17.3934,Z 58,A -102.1177,B 24.8264,C -3.0394,E1 24.9866,E2 -895.4514} C_DIS
LIN {X -0.5649,Y -17.4774,Z 58,A -98.023,B 24.8263,C -3.0399,E1 24.998,E2 -899.5483} C_DIS
LIN {X -0.5649,Y -17.4774,Z 58,A -98.023,B 24.8263,C -3.0399,E1 24.998,E2 -899.5483} C_DIS
Enddeposition()
LIN {X 0.0634,Y -16.5053,Z 58,A -98.2,B 24.8258,C -3.0443,E1 24.9976,E2 -899.3818} C_DIS
Startdeposition()
$VEL.CP = VEL_PRINT
LIN {X -1.6166,Y -16.4281,Z 58,A -103.8398,B 24.8257,C -3.0452,E1 24.9819,E2 -893.7422} C_DIS
LIN {X -2.7704,Y -16.2732,Z 58,A -108.1897,B 24.8257,C -3.0447,E1 24.9698,E2 -889.3871} C_DIS
LIN {X -4.3974,Y -15.9111,Z 58,A -114.7661,B 24.8258,C -3.0441,E1 24.952,E2 -882.8} C_DIS
LIN {X -6.7521,Y -15.0626,Z 58,A -122.615,B 24.8245,C -3.0558,E1 24.9317,E2 -874.9621} C_DIS
LIN {X -8.341,Y -14.2448,Z 58,A -128.9329,B 24.8236,C -3.0633,E1 24.9162,E2 -868.6443} C_DIS
LIN {X -9.6077,Y -13.4232,Z 58,A -134.1762,B 24.8226,C -3.0715,E1 24.9041,E2 -863.403} C_DIS
LIN {X -10.7635,Y -12.5151,Z 58,A -139.7435,B 24.8218,C -3.0792,E1 24.8921,E2 -857.8327} C_DIS
LIN {X -11.9882,Y -11.3453,Z 58,A -144.6873,B 24.82,C -3.0942,E1 24.8824,E2 -852.904} C_DIS
LIN {X -12.9223,Y -10.2717,Z 58,A -149.9625,B 24.8188,C -3.1042,E1 24.8729,E2 -847.6285} C_DIS
LIN {X -13.8313,Y -9.0105,Z 58,A -155.4288,B 24.8173,C -3.1171,E1 24.8642,E2 -842.1662} C_DIS
LIN {X -14.4183,Y -8.0376,Z 58,A -159.165,B 24.816,C -3.1279,E1 24.859,E2 -838.4362} C_DIS
LIN {X -14.9145,Y -7.0748,Z 58,A -163.0345,B 24.8149,C -3.1377,E1 24.8542,E2 -834.5694} C_DIS
LIN {X -15.4197,Y -5.893,Z 58,A -167.8106,B 24.8135,C -3.1494,E1 24.8492,E2 -829.7948} C_DIS
LIN {X -15.8481,Y -4.6189,Z 58,A -172.3128,B 24.8118,C -3.1633,E1 24.8454,E2 -825.3} C_DIS
LIN {X -16.1981,Y -3.178,Z 58,A -178.4197,B 24.8102,C -3.1766,E1 24.8418,E2 -819.189} C_DIS
LIN {X -16.4101,Y -1.7879,Z 58,A 176.7566,B 24.8084,C -3.1916,E1 24.8402,E2 -814.3725} C_DIS
LIN {X -16.5037,Y 0.3484,Z 58,A 170.0933,B 24.8054,C -3.2163,E1 24.8399,E2 -807.7281} C_DIS
LIN {X -16.4518,Y 1.3519,Z 58,A 165.5526,B 24.8044,C -3.2249,E1 24.8409,E2 -803.1809} C_DIS
LIN {X -16.0855,Y 3.7077,Z 58,A 158.2836,B 24.801,C -3.2526,E1 24.8445,E2 -795.9353} C_DIS
LIN {X -15.5958,Y 5.4098,Z 58,A 150.8039,B 24.7991,C -3.2683,E1 24.8509,E2 -788.4502} C_DIS
LIN {X -14.9821,Y 6.9303,Z 58,A 145.0024,B 24.797,C -3.2846,E1 24.8576,E2 -782.656} C_DIS
LIN {X -13.772,Y 9.1007,Z 58,A 137.286,B 24.7938,C -3.3106,E1 24.8686,E2 -774.9623} C_DIS
LIN {X -12.7494,Y 10.4852,Z 58,A 131.3288,B 24.7919,C -3.3261,E1 24.8788,E2 -769.0138} C_DIS
LIN {X -11.6394,Y 11.7049,Z 58,A 125.4355,B 24.7902,C -3.3392,E1 24.8901,E2 -763.1265} C_DIS
LIN {X -10.4184,Y 12.8043,Z 58,A 119.5999,B 24.7887,C -3.3511,E1 24.9025,E2 -757.2968} C_DIS
LIN {X -8.848,Y 13.9349,Z 58,A 113.0589,B 24.787,C -3.3646,E1 24.9176,E2 -750.7659} C_DIS
LIN {X -7.9672,Y 14.4575,Z 58,A 109.3224,B 24.7863,C -3.3699,E1 24.9267,E2 -747.0313} C_DIS
LIN {X -6.371,Y 15.2279,Z 58,A 103.9618,B 24.7848,C -3.3819,E1 24.9402,E2 -741.6863} C_DIS
LIN {X -5.2229,Y 15.6591,Z 58,A 99.2285,B 24.7844,C -3.3852,E1 24.9527,E2 -736.9515} C_DIS
LIN {X -3.9219,Y 16.0346,Z 58,A 94.4893,B 24.7838,C -3.3897,E1 24.9655,E2 -732.2158} C_DIS
LIN {X -2.7217,Y 16.2814,Z 58,A 90.3998,B 24.7833,C -3.3936,E1 24.9767,E2 -728.1314} C_DIS
LIN {X -1.5748,Y 16.4321,Z 58,A 86.2311,B 24.7831,C -3.395,E1 24.9882,E2 -723.9635} C_DIS
LIN {X -0.1144,Y 16.5069,Z 58,A 80.8748,B 24.7831,C -3.395,E1 25.0032,E2 -718.6066} C_DIS
LIN {X 1.3098,Y 16.4552,Z 58,A 75.3848,B 24.7835,C -3.3922,E1 25.0185,E2 -713.1121} C_DIS
LIN {X 3.7372,Y 16.0783,Z 58,A 67.9739,B 24.7831,C -3.3953,E1 25.0388,E2 -705.7169} C_DIS
LIN {X 4.9972,Y 15.7329,Z 58,A 63.0783,B 24.7837,C -3.3901,E1 25.0519,E2 -700.8171} C_DIS
LIN {X 6.1617,Y 15.3143,Z 58,A 58.4518,B 24.7845,C -3.384,E1 25.064,E2 -696.1863} C_DIS
LIN {X 7.7934,Y 14.5516,Z 58,A 53.0294,B 24.7848,C -3.3818,E1 25.0775,E2 -690.7733} C_DIS
LIN {X 8.9161,Y 13.8922,Z 58,A 48.1129,B 24.786,C -3.3726,E1 25.0893,E2 -685.8502} C_DIS
LIN {X 9.9958,Y 13.1371,Z 58,A 43.6266,B 24.7869,C -3.3656,E1 25.0994,E2 -681.3631} C_DIS
LIN {X 11.0318,Y 12.2797,Z 58,A 39.2174,B 24.7877,C -3.3587,E1 25.1087,E2 -676.9547} C_DIS
LIN {X 11.98,Y 11.3567,Z 58,A 34.1538,B 24.7894,C -3.3457,E1 25.1187,E2 -671.8819} C_DIS
LIN {X 13.1105,Y 10.0304,Z 58,A 28.663,B 24.7906,C -3.3362,E1 25.1284,E2 -666.3938} C_DIS
LIN {X 13.8682,Y 8.9535,Z 58,A 23.688,B 24.7924,C -3.3218,E1 25.1362,E2 -661.4093} C_DIS
LIN {X 14.611,Y 7.6818,Z 58,A 18.5099,B 24.7941,C -3.3079,E1 25.1432,E2 -656.2252} C_DIS
LIN {X 15.2907,Y 6.2196,Z 58,A 12.4313,B 24.7966,C -3.2885,E1 25.1499,E2 -650.1339} C_DIS
LIN {X 15.9919,Y 4.0923,Z 58,A 5.1697,B 24.7989,C -3.27,E1 25.1557,E2 -642.8698} C_DIS
LIN {X 16.3295,Y 2.4161,Z 58,A -0.6692,B 24.801,C -3.2528,E1 25.1586,E2 -637.0245} C_DIS
LIN {X 16.4894,Y 0.7703,Z 58,A -5.9924,B 24.8027,C -3.2386,E1 25.1597,E2 -631.6992} C_DIS
LIN {X 16.5028,Y -0.3914,Z 58,A -9.8359,B 24.8041,C -3.2277,E1 25.1597,E2 -627.8526} C_DIS
LIN {X 16.4038,Y -1.8466,Z 58,A -14.9997,B 24.8061,C -3.211,E1 25.1585,E2 -622.68} C_DIS
LIN {X 16.2339,Y -2.9927,Z 58,A -19.2182,B 24.8078,C -3.1969,E1 25.1565,E2 -618.4527} C_DIS
LIN {X 15.867,Y -4.5533,Z 58,A -24.7261,B 24.8098,C -3.1803,E1 25.1527,E2 -612.9373} C_DIS
LIN {X 15.4659,Y -5.771,Z 58,A -29.0161,B 24.8112,C -3.1683,E1 25.1487,E2 -608.6428} C_DIS
LIN {X 14.8442,Y -7.221,Z 58,A -35.3363,B 24.814,C -3.1454,E1 25.1413,E2 -602.3025} C_DIS
LIN {X 14.1835,Y -8.4444,Z 58,A -39.8558,B 24.8153,C -3.1343,E1 25.135,E2 -597.7801} C_DIS
LIN {X 13.0339,Y -10.1298,Z 58,A -46.1004,B 24.8167,C -3.1222,E1 25.1249,E2 -591.5371} C_DIS
LIN {X 11.9505,Y -11.3867,Z 58,A -52.6369,B 24.8191,C -3.1019,E1 25.1126,E2 -584.9817} C_DIS
LIN {X 10.4709,Y -12.7605,Z 58,A -60.2615,B 24.8214,C -3.0819,E1 25.0965,E2 -577.3395} C_DIS
LIN {X 9.1475,Y -13.7411,Z 58,A -64.6698,B 24.8216,C -3.0801,E1 25.0864,E2 -572.9421} C_DIS
LIN {X 8.2511,Y -14.2969,Z 58,A -68.158,B 24.8223,C -3.0748,E1 25.0781,E2 -569.452} C_DIS
LIN {X 7.058,Y -14.9225,Z 58,A -73.1577,B 24.8234,C -3.0651,E1 25.0656,E2 -564.4428} C_DIS
LIN {X 5.5885,Y -15.5327,Z 58,A -77.9235,B 24.8237,C -3.0627,E1 25.0532,E2 -559.682} C_DIS
LIN {X 4.5961,Y -15.8548,Z 58,A -82.4691,B 24.8248,C -3.0526,E1 25.0411,E2 -555.1205} C_DIS
LIN {X 3.3584,Y -16.1621,Z 58,A -87.0945,B 24.8254,C -3.0474,E1 25.0284,E2 -550.4889} C_DIS
LIN {X 1.3233,Y -16.4542,Z 58,A -93.0266,B 24.8251,C -3.0502,E1 25.012,E2 -544.5681} C_DIS
LIN {X 0.0634,Y -16.5053,Z 58,A -98.2,B 24.8258,C -3.0443,E1 24.9976,E2 -539.3818} C_DIS
Enddeposition()
LIN {X 0.0634,Y -16.5053,Z 58,A -98.2,B 24.8258,C -3.0443,E1 24.9976,E2 -539.3818} C_DIS
Startdeposition()
$VEL.CP = VEL_PRINT
LIN {X 0.5689,Y -15.5179,Z 58,A -94.3173,B 24.8225,C -3.0729,E1 25.0086,E2 -543.332} C_DIS
LIN {X 2.2141,Y -15.3693,Z 58,A -88.2703,B 24.8221,C -3.076,E1 25.0254,E2 -549.3823} C_DIS
LIN {X 3.2854,Y -15.1766,Z 58,A -83.1821,B 24.821,C -3.0859,E1 25.0394,E2 -554.4877} C_DIS
LIN {X 5.1761,Y -14.6401,Z 58,A -76.3824,B 24.8203,C -3.0913,E1 25.0574,E2 -561.288} C_DIS
LIN {X 6.5144,Y -14.0938,Z 58,A -71.7516,B 24.82,C -3.0944,E1 25.0693,E2 -565.9149} C_DIS
LIN {X 7.5598,Y -13.5637,Z 58,A -67.2185,B 24.819,C -3.1029,E1 25.0805,E2 -570.4555} C_DIS
LIN {X 8.5753,Y -12.9456,Z 58,A -62.9642,B 24.8181,C -3.1101,E1 25.0906,E2 -574.7132} C_DIS
LIN {X 9.8444,Y -12.0082,Z 58,A -56.374,B 24.816,C -3.1278,E1 25.1051,E2 -581.3213} C_DIS
LIN {X 11.2442,Y -10.7088,Z 58,A -48.9836,B 24.8138,C -3.147,E1 25.1198,E2 -588.7259} C_DIS
LIN {X 12.3939,Y -9.3549,Z 58,A -42.8405,B 24.8122,C -3.1606,E1 25.1305,E2 -594.8727} C_DIS
LIN {X 13.2919,Y -8.0281,Z 58,A -37.4035,B 24.8107,C -3.173,E1 25.1387,E2 -600.3117} C_DIS
LIN {X 13.9689,Y -6.782,Z 58,A -32.1803,B 24.8089,C -3.188,E1 25.1453,E2 -605.5427} C_DIS
LIN {X 14.483,Y -5.6008,Z 58,A -27.5352,B 24.8073,C -3.2012,E1 25.1503,E2 -610.1934} C_DIS
LIN {X 14.9447,Y -4.2165,Z 58,A -21.7955,B 24.8049,C -3.2204,E1 25.155,E2 -615.9461} C_DIS
LIN {X 15.3597,Y -2.2824,Z 58,A -14.0117,B 24.8017,C -3.2471,E1 25.1588,E2 -623.7475} C_DIS
LIN {X 15.5261,Y -0.2537,Z 58,A -7.9315,B 24.8003,C -3.2586,E1 25.1598,E2 -629.8188} C_DIS
LIN {X 15.4841,Y 1.1703,Z 58,A -2.3446,B 24.7979,C -3.2776,E1 25.1591,E2 -635.4176} C_DIS
LIN {X 15.3325,Y 2.4558,Z 58,A 2.1966,B 24.7964,C -3.2902,E1 25.1573,E2 -639.9619} C_DIS
LIN {X 14.8958,Y 4.386,Z 58,A 10.5903,B 24.7925,C -3.3207,E1 25.1516,E2 -648.3796} C_DIS
LIN {X 14.3044,Y 6.042,Z 58,A 16.4187,B 24.7909,C -3.3337,E1 25.1456,E2 -654.2065} C_DIS
LIN {X 13.6629,Y 7.3743,Z 58,A 21.2505,B 24.7897,C -3.3435,E1 25.1396,E2 -659.0357} C_DIS
LIN {X 12.8923,Y 8.6553,Z 58,A 27.4466,B 24.7873,C -3.3625,E1 25.1303,E2 -665.2458} C_DIS
LIN {X 12.0631,Y 9.7777,Z 58,A 32.108,B 24.7862,C -3.3709,E1 25.1223,E2 -669.905} C_DIS
LIN {X 11.1238,Y 10.8346,Z 58,A 37.3228,B 24.7848,C -3.382,E1 25.1124,E2 -675.1235} C_DIS
LIN {X 10.233,Y 11.6794,Z 58,A 41.9499,B 24.7835,C -3.3915,E1 25.1029,E2 -679.7545} C_DIS
LIN {X 9.1269,Y 12.5628,Z 58,A 47.0739,B 24.7825,C -3.3999,E1 25.0915,E2 -684.8796} C_DIS
LIN {X 7.7349,Y 13.4642,Z 58,A 53.4254,B 24.7811,C -3.4104,E1 25.0764,E2 -691.236} C_DIS
LIN {X 6.4501,Y 14.1253,Z 58,A 58.6199,B 24.7804,C -3.4158,E1 25.0634,E2 -696.4297} C_DIS
LIN {X 5.0472,Y 14.685,Z 58,A 64.5554,B 24.7795,C -3.423,E1 25.0478,E2 -702.3698} C_DIS
LIN {X 3.4417,Y 15.1418,Z 58,A 70.437,B 24.7792,C -3.4249,E1 25.0319,E2 -708.2472} C_DIS
LIN {X 1.9786,Y 15.4015,Z 58,A 75.2675,B 24.7795,C -3.423,E1 25.0186,E2 -713.0685} C_DIS
LIN {X 0.9762,Y 15.4975,Z 58,A 80.4092,B 24.7785,C -3.4305,E1 25.0042,E2 -718.2255} C_DIS
LIN {X -1.1608,Y 15.4846,Z 58,A 87.2799,B 24.7795,C -3.4232,E1 24.9851,E2 -725.08} C_DIS
LIN {X -2.4434,Y 15.3344,Z 58,A 93.1243,B 24.7792,C -3.425,E1 24.969,E2 -730.9336} C_DIS
LIN {X -4.7731,Y 14.7763,Z 58,A 100.6453,B 24.7811,C -3.4108,E1 24.9488,E2 -738.4319} C_DIS
LIN {X -6.0588,Y 14.2974,Z 58,A 106.5086,B 24.7815,C -3.4071,E1 24.9335,E2 -744.2992} C_DIS
LIN {X -7.1937,Y 13.7612,Z 58,A 110.7291,B 24.7827,C -3.3984,E1 24.923,E2 -748.5102} C_DIS
Enddeposition()
END
